Omron CX-Programmer project NewProject (CX-Programmer 9.74)

# PLC M1: CJ2M CPU32
I/O table (CPU CJ2M-CPU32): rack 0 slot 0 CJ1W-ID211; rack 0 slot 1 CJ1W-ID211; rack 0 slot 2 CJ1W-OD212; rack 0 slot 3 CJ1W-OC211; rack 0 slot 4 CJ1W-TC104; rack 0 slot 11 CJ2M-EIP21

## Data types
TYPE s_maquina_in : STRUCT  (* Inputs da maquina *)
  st_ciclo : BOOL;  (* Botão inicio de ciclo *)
  sp_ciclo : BOOL;  (* Botão fim de ciclo *)
  sel_carga : BOOL;  (* Botão selecção de carga *)
  st_carga : BOOL;  (* Botão inicio de carga *)
  fcf_carga : BOOL;  (* Fim de curso fechado carga *)
  sel_dcarga : BOOL;  (* Botão selecção de descarga *)
  st_dcarga : BOOL;  (* Botão inicio de descarga *)
  fcf_dcarga : BOOL;  (* Fim de curso fechado descarga *)
  psl : BOOL;  (* Pressostato *)
  nhrz : BOOL;  (* Maquina não horizontal *)
  pe1 : BOOL;  (* Paragem de emergência *)
  pe2 : BOOL;  (* Relé de segurança *)
  de : BOOL;  (* Disparo termico *)
  x0_13 : BOOL;  (* RESERVA *)
  x0_14 : BOOL;  (* RESERVA *)
  x0_15 : BOOL;  (* RESERVA *)
END_STRUCT END_TYPE
TYPE s_maquina_out : STRUCT  (* Outputs da maquina *)
  x0_0 : BOOL;  (* RESERVA *)
  x0_1 : BOOL;  (* RESERVA *)
  oma_carga : BOOL;  (* Abrir carga *)
  omf_carga : BOOL;  (* Fechar carga *)
  oma_dcarga : BOOL;  (* Abrir descarga *)
  omf_dcarga : BOOL;  (* Fechar descarga *)
  ok_carga : BOOL;  (* Carga confirmada (carregar rolhas) *)
  ok_dcarga : BOOL;  (* Descarga confirmada (descarregar rolhas) *)
  x0_8 : BOOL;  (* RESERVA *)
  x0_9 : BOOL;  (* RESERVA *)
  x0_10 : BOOL;  (* RESERVA *)
  x0_11 : BOOL;  (* RESERVA *)
  x0_12 : BOOL;  (* RESERVA *)
  x0_13 : BOOL;  (* RESERVA *)
  x0_14 : BOOL;  (* RESERVA *)
  x0_15 : BOOL;  (* RESERVA *)
END_STRUCT END_TYPE
TYPE s_maquina_lmp : STRUCT  (* Lampadas da maquina *)
  oms_inicio : BOOL;  (* Lampada inicio *)
  oms_carga : BOOL;  (* Lampada carga *)
  oms_dcarga : BOOL;  (* Lampada descarga *)
  x0_3 : BOOL;  (* RESERVA *)
  x0_4 : BOOL;  (* RESERVA *)
  x0_5 : BOOL;  (* RESERVA *)
  x0_6 : BOOL;  (* RESERVA *)
  x0_7 : BOOL;  (* RESERVA *)
  oms_red : BOOL;  (* Lampada FLASH vermelho *)
  oms_green : BOOL;  (* Lampada FLASH verde *)
  x0_10 : BOOL;  (* RESERVA *)
  x0_11 : BOOL;  (* RESERVA *)
  x0_12 : BOOL;  (* RESERVA *)
  x0_13 : BOOL;  (* RESERVA *)
  oms_ilum : BOOL;  (* Iluminação *)
  alm : BOOL;  (* Maquina em alarme (Alarmes que não páram a maquina) *)
END_STRUCT END_TYPE
TYPE s_maquina_defs : STRUCT  (* Defeitos da maquina *)
  def1 : BOOL;  (* Paragem de emergência *)
  def2 : BOOL;  (* Relé de segurança *)
  def3 : BOOL;  (* Disparo termico *)
  def4 : BOOL;  (* RESERVA *)
  def5 : BOOL;  (* Defeito de aspiração *)
  def6 : BOOL;  (* Defeito de tratamento *)
  def7 : BOOL;  (* Defeito de injecção *)
  def8 : BOOL;  (* Defeito de aquecimento *)
  def9 : BOOL;  (* Maquina não horizontal *)
  def10 : BOOL;  (* Pressão de ar baixa *)
  def11 : BOOL;  (* RESERVA *)
  def12 : BOOL;  (* RESERVA *)
  def13 : BOOL;  (* RESERVA *)
  def14 : BOOL;  (* RESERVA *)
  def15 : BOOL;  (* Falha de manobra na carga *)
  def16 : BOOL;  (* Falha de manobra na descarga *)
END_STRUCT END_TYPE
TYPE s_maquina_bits : STRUCT  (* Bits auxiliares da maquina *)
  rst : BOOL;  (* Reset aos defeitos *)
  dgm : BOOL;  (* Defeito geral *)
  mdp : BOOL;  (* Maquina disponivel *)
  x0_3 : BOOL;  (* RESERVA *)
  x0_4 : BOOL;  (* RESERVA *)
  x0_5 : BOOL;  (* RESERVA *)
  x0_6 : BOOL;  (* RESERVA *)
  x0_7 : BOOL;  (* RESERVA *)
  dp_tcarga : BOOL;  (* Transporte de carga disponivel (Maquina permite fazer transporte de carga) *)
  om_carga : BOOL;  (* Abrir carga *)
  om_dcarga : BOOL;  (* Abrir descarga *)
  LockDescarga : BOOL;  (* Bloquear descarga *)
  x0_12 : BOOL;  (* RESERVA *)
  x0_13 : BOOL;  (* RESERVA *)
  x0_14 : BOOL;  (* RESERVA *)
  x0_15 : BOOL;  (* RESERVA *)
  x1_0 : BOOL;  (* RESERVA *)
  x1_1 : BOOL;  (* RESERVA *)
  x1_2 : BOOL;  (* RESERVA *)
  x1_3 : BOOL;  (* RESERVA *)
  x1_4 : BOOL;  (* RESERVA *)
  x1_5 : BOOL;  (* RESERVA *)
  x1_6 : BOOL;  (* RESERVA *)
  inj_block : BOOL;  (* Injecção bloqueada *)
  act_ciclo : BOOL;  (* Ciclo - Activo *)
  om_ciclo : BOOL;  (* Ciclo - Ordem de marcha *)
  new_of : BOOL;  (* Nova ordem de fabrico *)
  val_ciclo : BOOL;  (* Ciclo validado pelo MES *)
  com_fail : BOOL;  (* Falha de comunicação com o MES *)
  st_mes : BOOL;  (* Arranque da ordem com MES *)
  x1_14 : BOOL;  (* RESERVA *)
  new_man : BOOL;  (* Nova ordem manual *)
END_STRUCT END_TYPE
TYPE s_maquina_hmi : STRUCT  (* Dados do HMI *)
  st_ciclo : BOOL;  (* Botão inicio de ciclo *)
  sp_ciclo : BOOL;  (* Botão fim de ciclo *)
  sel_carga : BOOL;  (* Botão selecção de carga *)
  st_carga : BOOL;  (* Botão inicio de carga *)
  sel_dcarga : BOOL;  (* Botão selecção de descarga *)
  st_dcarga : BOOL;  (* Botão inicio de descarga *)
  on_msg : BOOL;  (* Mostra janela de mensagens *)
  x0_7 : BOOL;  (* RESERVA *)
  x0_8 : BOOL;  (* RESERVA *)
  x0_9 : BOOL;  (* RESERVA *)
  x0_10 : BOOL;  (* RESERVA *)
  x0_11 : BOOL;  (* RESERVA *)
  x0_12 : BOOL;  (* RESERVA *)
  x0_13 : BOOL;  (* RESERVA *)
  x0_14 : BOOL;  (* RESERVA *)
  x0_15 : BOOL;  (* RESERVA *)
END_STRUCT END_TYPE
TYPE s_maquina : STRUCT  (* Dados da maquina *)
  modo : INT;  (* Modo de funcionamento (0-Manual, 1-Offline, 2-Online) *)
  etapa : INT;  (* Etapa actual (10-Carga, 20-Tratamento, 30-Descarga) *)
  in : s_maquina_in;  (* Entradas *)
  out : s_maquina_out;  (* Saidas *)
  hmi : s_maquina_hmi;  (* Dados do HMI *)
  bits : s_maquina_bits;  (* Bits auxiliares *)
  lmp : s_maquina_lmp;  (* Lampadas *)
  def : s_maquina_defs;  (* Defeitos *)
  cp_mes : s_maquina_mes;  (* Causas de paragem do MES *)
  log : s_maq_log;  (* Dados de datalogger *)
  pss_exe : s_pss_exe;  (* Passo actual a executar *)
  modo_hmi : INT;  (* Valor colocado pelo operador *)
  cparagem : INT;  (* Causa de paragem *)
  num_msg : INT;  (* Numero da mensagem *)
  rsv2 : INT Dimensions=[17];  (* RESERVA *)
  pt_sb : INT Dimensions=[5];  (* Zona SB da consola *)
  pt_sw : INT Dimensions=[5];  (* Zona SW da consola *)
END_STRUCT END_TYPE
TYPE s_f_aspira : STRUCT  (* Dados da função aspiração *)
  fca : BOOL;  (* Aspiração aberta *)
  fcf : BOOL;  (* Aspiração fechada *)
  oma : BOOL;  (* Abrir aspiração *)
  omf : BOOL;  (* Fechar aspiração *)
  rm : BOOL;  (* Resposta de marcha do ventilador de aspiração *)
  fm : BOOL;  (* Falha de manobra na aspiração *)
  fmv : BOOL;  (* Falha do ventilador de aspiração *)
  om_aquece : BOOL;  (* Aquecimento em curso (Pede aspiração) *)
  on : BOOL;  (* Aspiração em marcha e ok *)
  x0_9 : BOOL;  (* RESERVA *)
  x0_10 : BOOL;  (* RESERVA *)
  x0_11 : BOOL;  (* RESERVA *)
  x0_12 : BOOL;  (* RESERVA *)
  st_hmi : BOOL;  (* Arranque do hmi *)
  sp_hmi : BOOL;  (* Paragem do hmi *)
  cfm : BOOL;  (* Condição de funcionamento manual *)
  es : INT;  (* Estado *)
  rsv1 : INT Dimensions=[16];  (* RESERVA *)
  tt : REAL;  (* Totalizador *)
END_STRUCT END_TYPE
TYPE s_tc104_cio : STRUCT  (* Dados CIO da carta TC104 *)
  sp1 : INT;  (* Loop 1 Set Point (SP) *)
  sp2 : INT;  (* Loop 2 Set Point (SP) *)
  l2_st_at : BOOL;  (* Loop 2 Start AT *)
  l2_sp_at : BOOL;  (* Loop 2 Stop AT *)
  l1_st_at : BOOL;  (* Loop 1 Start AT *)
  l1_sp_at : BOOL;  (* Loop 1 Stop AT *)
  l2_sp : BOOL;  (* Loop 2 Stop *)
  x2_5 : BOOL;  (* RESERVA *)
  l1_sp : BOOL;  (* Loop 1 Stop *)
  x2_7 : BOOL;  (* RESERVA *)
  x2_8 : BOOL;  (* RESERVA *)
  x2_9 : BOOL;  (* RESERVA *)
  x2_10 : BOOL;  (* RESERVA *)
  x2_11 : BOOL;  (* RESERVA *)
  l2_ch_pid_c : BOOL;  (* Loop 2 Change PID Constants *)
  l1_ch_pid_c : BOOL;  (* Loop 1 Change PID Constants *)
  l2_save : BOOL;  (* Loop 2 Save *)
  l1_save : BOOL;  (* Loop 1 Save *)
  pv1 : INT;  (* Loop 1 PV *)
  pv2 : INT;  (* Loop 2 PV *)
  sp1_r : INT;  (* Loop 1 Set Point (SP) - Read *)
  sp2_r : INT;  (* Loop 2 Set Point (SP) - Read *)
  l1_l2_dp_err : WORD;  (* Loop 1/2 Decimal point & error number *)
  l1_s_al2 : BOOL;  (* Loop 1 - Status AL2 *)
  l1_s_al1 : BOOL;  (* Loop 1 - Status AL1 *)
  l1_s_hb : BOOL;  (* Loop 1 - Status HB *)
  l1_s_at : BOOL;  (* Loop 1 - Status AT *)
  l1_s_ctrlout : BOOL;  (* Loop 1 - Status Control Output *)
  x8_5 : BOOL;  (* RESERVA *)
  x8_6 : BOOL;  (* RESERVA *)
  x8_7 : BOOL;  (* RESERVA *)
  l1_s_sp : BOOL;  (* Loop 1 - Status Stop *)
  l1_s_err : BOOL;  (* Loop 1 - Status Setting Error *)
  l1_s_pid_calc : BOOL;  (* Loop 1 - Status PID Constants Calculated *)
  l1_s_sby : BOOL;  (* Loop 1 - Status Standby *)
  l1_s_ferr : BOOL;  (* Loop 1 - Status Fatal Error *)
  l1_s_ct_ovf : BOOL;  (* Loop 1 - Status Overflow *)
  l1_s_serr : BOOL;  (* Loop 1 - Status Sensor Error *)
  l1_s_savec : BOOL;  (* Loop 1 - Status Save Completed *)
  l2_s_al2 : BOOL;  (* Loop 2 - Status AL2 *)
  l2_s_al1 : BOOL;  (* Loop 2 - Status AL1 *)
  l2_s_hb : BOOL;  (* Loop 2 - Status HB *)
  l2_s_at : BOOL;  (* Loop 2 - Status AT *)
  l2_s_ctrlout : BOOL;  (* Loop 2 - Status Control Output *)
  x9_5 : BOOL;  (* RESERVA *)
  x9_6 : BOOL;  (* RESERVA *)
  x9_7 : BOOL;  (* RESERVA *)
  l2_s_sp : BOOL;  (* Loop 2 - Status Stop *)
  l2_s_err : BOOL;  (* Loop 2 - Status Setting Error *)
  l2_s_pid_calc : BOOL;  (* Loop 2 - Status PID Constants Calculated *)
  l2_s_sby : BOOL;  (* Loop 2 - Status Standby *)
  l2_s_ferr : BOOL;  (* Loop 2 - Status Fatal Error *)
  l2_s_ct_ovf : BOOL;  (* Loop 2 - Status Overflow *)
  l2_s_serr : BOOL;  (* Loop 2 - Status Sensor Error *)
  l2_s_savec : BOOL;  (* Loop 2 - Status Save Completed *)
  hb_sp1 : INT;  (* Loop 1 - Heater Burnout Set Value *)
  hb_sp2 : INT;  (* Loop 2 - Heater Burnout Set Value *)
  rsv1 : INT;  (* RESERVA *)
  hc1 : INT;  (* Loop 1 - Heater Current *)
  hc2 : INT;  (* Loop 2 - Heater Current *)
  hb_sp1_r : INT;  (* Loop 1 - Heater Burnout Set Value - Read *)
  hb_sp2_r : INT;  (* Loop 2 - Heater Burnout Set Value - Read *)
  rsv2 : INT Dimensions=[3];  (* RESERVA *)
END_STRUCT END_TYPE
TYPE s_tc104_dm : STRUCT  (* Dados DM da carta TC104 *)
  dados : INT Dimensions=[100];  (* Dados da carta *)
END_STRUCT END_TYPE
TYPE s_f_aquece : STRUCT  (* Dados da função aquecimento *)
  rm_r : BOOL;  (* Contactor das resistências *)
  rm_v : BOOL;  (* Resposta de marcha do ventilador *)
  ok_fx : BOOL;  (* Detector de fluxo OK *)
  x0_3 : BOOL;  (* RESERVA *)
  ft : BOOL;  (* Falha de temperatura *)
  ini : BOOL;  (* Inicio do aquecimento *)
  ini_tt : BOOL;  (* Inicio da contagem do tempo *)
  ok_sp : BOOL;  (* Dentro da vizinhaça de setpoint a controlar *)
  om : BOOL;  (* Ordem de marcha para aquecimento *)
  fm_r : BOOL;  (* Falha de marcha das resistências *)
  fm_v : BOOL;  (* Falha de marcha do ventilador *)
  fm_fx : BOOL;  (* Falha no detector de fluxo *)
  fm_a : BOOL;  (* Falha na aspiração *)
  st_hmi : BOOL;  (* Arranque do hmi *)
  sp_hmi : BOOL;  (* Paragem do hmi *)
  cfm : BOOL;  (* Condição de funcionamento manual *)
  es_r : INT;  (* Estado *)
  sp : REAL;  (* Setpoint de temperatura *)
  pv : REAL;  (* Temperatura actual *)
  sp_delta : REAL;  (* Valor de vizinhança apartir do qual começa a contar tempo de aquecimento *)
  sp_ft : INT;  (* Tempo para dar falha de temperatura *)
  es_v : INT;  (* Estado *)
  rsv2 : INT Dimensions=[8];  (* RESERVA *)
  tt : REAL;  (* Totalizador *)
END_STRUCT END_TYPE
TYPE s_f_trata : STRUCT  (* Dados da função tratamento *)
  rm : BOOL;  (* Marcha do tambor *)
  om1 : BOOL;  (* Ordem de marcha 1 *)
  om2 : BOOL;  (* Ordem de marcha 2 *)
  omx : BOOL;  (* Ordem de marcha auxiliar *)
  fm : BOOL;  (* Falha de marcha do tambor *)
  x0_5 : BOOL;  (* RESERVA *)
  x0_6 : BOOL;  (* RESERVA *)
  x0_7 : BOOL;  (* RESERVA *)
  x0_8 : BOOL;  (* RESERVA *)
  x0_9 : BOOL;  (* RESERVA *)
  x0_10 : BOOL;  (* RESERVA *)
  x0_11 : BOOL;  (* RESERVA *)
  x0_12 : BOOL;  (* RESERVA *)
  x0_13 : BOOL;  (* RESERVA *)
  x0_14 : BOOL;  (* RESERVA *)
  cfm : BOOL;  (* Condição de funcionamento manual *)
  es : INT;  (* Estado *)
  rsv2 : INT Dimensions=[16];  (* RESERVA *)
  tt : REAL;  (* Totalizador *)
END_STRUCT END_TYPE
TYPE s_f_injecta : STRUCT  (* Dados da função injecção *)
  x0_0 : BOOL;  (* RESERVA *)
  x0_1 : BOOL;  (* RESERVA *)
  om1 : BOOL;  (* Ordem de marcha *)
  om2 : BOOL;  (* Ordem de marcha spray *)
  finj : BOOL;  (* Falha de injecção *)
  fg : BOOL;  (* Fuga de produto *)
  x0_6 : BOOL;  (* RESERVA *)
  s_insp : BOOL;  (* Inspecção activada *)
  inj : BOOL;  (* Pede permissão para injectar *)
  inj_ok : BOOL;  (* Recebe autorização para injectar *)
  x0_10 : BOOL;  (* RESERVA *)
  x0_11 : BOOL;  (* RESERVA *)
  x0_12 : BOOL;  (* RESERVA *)
  x0_13 : BOOL;  (* RESERVA *)
  cal : BOOL;  (* Calibração *)
  cfm : BOOL;  (* Condição de funcionamento manual *)
  es : INT;  (* Estado *)
  prod : INT;  (* Produto *)
  rsv1 : INT Dimensions=[15];  (* RESERVA *)
  tt : REAL;  (* Totalizador *)
END_STRUCT END_TYPE
TYPE s_caudal : STRUCT  (* Dados do caudalimetro *)
  tti : BOOL;  (* Impulso de totalização *)
  rst : BOOL;  (* Reset *)
  prod_used : BOOL;  (* Produto em uso *)
  fgp : BOOL;  (* Fuga de produto *)
  ftt : BOOL;  (* Falha de caudal *)
  rem : BOOL;  (* Totalizador local/remoto *)
  rem_ok : BOOL;  (* OK para ir buscar o valor do totalizador remoto *)
  inj_ini : BOOL;  (* Inicio da injecção *)
  x0_8 : BOOL;  (* RESERVA *)
  x0_9 : BOOL;  (* RESERVA *)
  x0_10 : BOOL;  (* RESERVA *)
  x0_11 : BOOL;  (* RESERVA *)
  x0_12 : BOOL;  (* RESERVA *)
  x0_13 : BOOL;  (* RESERVA *)
  x0_14 : BOOL;  (* RESERVA *)
  x0_15 : BOOL;  (* RESERVA *)
  prod : INT;  (* Produto *)
  rsv1 : INT Dimensions=[6];  (* RESERVA *)
  tti_x : REAL;  (* Valor do impulso *)
  tt_rem : REAL;  (* Totalizador remoto *)
  tt_rem_old : REAL;  (* Totalizador remoto antigo *)
  tt_inj : REAL;  (* Totalizador de injecção *)
  tt_p : REAL;  (* Totalizador parcial *)
  tt_g : REAL;  (* Totalizador global *)
END_STRUCT END_TYPE
TYPE s_carro : STRUCT  (* Dados do carro de injecção *)
  fcr : BOOL;  (* Fim de curso recuado *)
  fca : BOOL;  (* Fim de curso avanço *)
  oma : BOOL;  (* Ordem de marcha avanço *)
  omr : BOOL;  (* Ordem de marcha recuar *)
  omv : BOOL;  (* Ordem de marcha velocidade lenta *)
  fm : BOOL;  (* Falha de manobra *)
  av : BOOL;  (* Avaria *)
  i_pos : BOOL;  (* Impulsos de posição *)
  inj : BOOL;  (* Recebe pedido para injectar *)
  inj_ok : BOOL;  (* Informa que pode injectar *)
  cal : BOOL;  (* Calibrar *)
  src : BOOL;  (* Sentido recuar *)
  dgm : BOOL;  (* Defeito geral de maquina *)
  rm : BOOL;  (* Resposta de marcha *)
  cfma : BOOL;  (* Condição de funcionamento manual avançar *)
  cfmr : BOOL;  (* Condição de funcionamento manual recuar *)
  fav : BOOL;  (* Falha por avaria *)
  s_dp : BOOL;  (* Carrinho habilitado *)
  inj_cal : BOOL;  (* Calibração da injecção *)
  s_aut : BOOL;  (* Automatico *)
  x1_4 : BOOL;  (* RESERVA *)
  x1_5 : BOOL;  (* RESERVA *)
  x1_6 : BOOL;  (* RESERVA *)
  x1_7 : BOOL;  (* RESERVA *)
  x1_8 : BOOL;  (* RESERVA *)
  x1_9 : BOOL;  (* RESERVA *)
  x1_10 : BOOL;  (* RESERVA *)
  x1_11 : BOOL;  (* RESERVA *)
  x1_12 : BOOL;  (* RESERVA *)
  x1_13 : BOOL;  (* RESERVA *)
  x1_14 : BOOL;  (* RESERVA *)
  x1_15 : BOOL;  (* RESERVA *)
  rsv1 : INT Dimensions=[10];  (* RESERVA *)
  sp_min : REAL;  (* Setpoint posição minima de injecção *)
  sp_max : REAL;  (* Setpoint posição maxima de injecção *)
  pos_act : REAL;  (* Posição actual *)
  tt_i_act : INT;  (* Numero de impulsos actuais *)
  tt_i_max : INT;  (* Numero de impulsos maximos *)
END_STRUCT END_TYPE
TYPE s_of_cliente : STRUCT  (* Dados do cliente de uma OF *)
  nome : WORD Dimensions=[25];  (* Nome do cliente *)
  data : WORD Dimensions=[10];  (* Data de entrega *)
  produto : WORD Dimensions=[20];  (* Nome do produto *)
  prg_on : WORD Dimensions=[5];  (* Numero do programa online *)
  n_enc : WORD Dimensions=[10];  (* Numero de encomenda *)
  n_of : WORD Dimensions=[10];  (* Numero da OF *)
  n_lt : WORD Dimensions=[10];  (* Numero do lote *)
END_STRUCT END_TYPE
TYPE s_of_totais : STRUCT  (* Totais produzidos e a produzir de uma OF *)
  tt_global : UDINT;  (* Total a produzir na OF *)
  tt_falta : UDINT;  (* Total que falta produzir na OF *)
  tt_produzir : UDINT;  (* Total a produzir na maquina no batch *)
END_STRUCT END_TYPE
TYPE s_of_calibre : STRUCT  (* Calibre das rolhas a usar na OF *)
  dmt1 : REAL;  (* Diametro da rolha *)
  dmt2 : REAL;  (* Diametro da rolha *)
  h : REAL;  (* Comprimento da rolha *)
  a : REAL;  (* Area da rolha *)
  qtp : REAL;  (* Quantidade de produto *)
  cl_txt : WORD Dimensions=[10];  (* Calibre - Texto *)
END_STRUCT END_TYPE
TYPE s_of_pss : STRUCT  (* Passo individual do programa a executar *)
  f : INT;  (* Função *)
  p1 : INT;  (* Parametro 1 *)
  p2 : REAL;  (* Parametro 2 *)
  tt : REAL;  (* Totalizador *)
  uni : INT;  (* Unidade do totalizador *)
  rsv : INT Dimensions=[3];  (* RESERVA *)
END_STRUCT END_TYPE
TYPE s_of_prg : STRUCT  (* Programa a ser executado *)
  pss : s_of_pss Dimensions=[12];  (* Passos do programa a executar *)
END_STRUCT END_TYPE
TYPE s_of : STRUCT  (* Ordem de fabrico *)
  cliente : s_of_cliente;  (* Cliente da OF *)
  totais : s_of_totais;  (* Totais da OF *)
  calibre : s_of_calibre;  (* Calibre das rolhas da OF *)
  dados : BOOL;  (* OF com valores *)
  online : BOOL;  (* Ordem com dados para funcionar online *)
  nprg_off : INT;  (* Numero do programa offline *)
  rsv1 : INT Dimensions=[8];  (* RESERVA *)
  prg : s_of_prg;  (* Programa *)
END_STRUCT END_TYPE
TYPE s_pss_exe : STRUCT  (* Passo a executar *)
  pss : s_of_pss;  (* Passo actual a executar *)
  num_pss : INT;  (* Numero do passo actual *)
  ini : BOOL;  (* Inicio - Inicio do passo (Função faz inicializações necessárias) *)
  exe : BOOL;  (* Executar - Condição para funcionar (Função actua se valor igual a 1) *)
  fim : BOOL;  (* Fim - Terminado o passo (Função indica que terminou de executar) *)
  exc : BOOL;  (* Exclusivo - Condição para funções exclusivas (Função exclusiva coloca a 0 ao executar, impedindo que outras o façam) *)
  log : BOOL;  (* Fazer log *)
  rsv1 : INT Dimensions=[8];  (* RESERVA *)
END_STRUCT END_TYPE
TYPE s_mes_com : STRUCT  (* Comunicação com o MES *)
  n_enc : WORD Dimensions=[10];  (* Numero de encomenda *)
  n_of : WORD Dimensions=[10];  (* Numero da OF *)
  n_lt : WORD Dimensions=[10];  (* Numero do lote *)
  user : WORD Dimensions=[10];  (* Codigo do operador *)
  rsv1 : INT;  (* RESERVA *)
  mes_plc : INT;  (* Variável de verificação de comunicação do MES para o PLC *)
  mes_plcx : INT;  (* Variável de verificação de comunicação do MES para o PLC (Auxiliar) *)
  plc_mes : INT;  (* Variável de verificação de comunicação do PLC para o MES *)
  mes_com_fail : BOOL;  (* Falha de comunicação com o MES *)
  f_in_exe : INT;  (* Função a executar *)
  f_out_exe : INT;  (* Função executada *)
  new_of : INT;  (* Contador de nova OF *)
  ctrl_com_plc : INT;  (* Controlo da comunicação - Escrita do PLC *)
  ctrl_com_mes : INT;  (* Controlo da comunicação - Escrita do MES *)
END_STRUCT END_TYPE
TYPE s_maq_log : STRUCT  (* Dados de datalogger da maquina *)
  n_of : WORD Dimensions=[10];  (* Numero da OF *)
  user : WORD Dimensions=[10];  (* Codigo do operador *)
  pss_exe : s_pss_exe;  (* Dados do passo actual *)
END_STRUCT END_TYPE
TYPE s_maquina_mes : STRUCT  (* Causas de paragem para o MES *)
  cp8 : BOOL;  (* Problemas de caudal *)
  cp9 : BOOL;  (* Filtro entupido *)
  cp10 : BOOL;  (* Bomba desligada *)
  cp11 : BOOL;  (* Obstrução da linha *)
  cp6 : BOOL;  (* Alarme de aquecimento *)
  cp13 : BOOL;  (* Falha de sonda *)
  cp19 : BOOL;  (* Descarga sem tratamento *)
  cp5 : BOOL;  (* Falta de tensão *)
  cp15 : BOOL;  (* Fuga de produto *)
  cp18 : BOOL;  (* Baixa temperatura *)
  cp7 : BOOL;  (* Falha geral *)
  X0_11 : BOOL;  (* RESERVA *)
  x0_12 : BOOL;  (* RESERVA *)
  x0_13 : BOOL;  (* RESERVA *)
  x0_14 : BOOL;  (* RESERVA *)
  x0_15 : BOOL;  (* RESERVA *)
END_STRUCT END_TYPE
TYPE s_equip_ios : STRUCT  (* Equipamento - Entradas *)
  om : BOOL;  (* Ordem de marcha *)
  oma : BOOL;  (* Ordem de abrir *)
  omf : BOOL;  (* Ordem de fechar *)
  rm : BOOL;  (* Resposta de marcha *)
  fca : BOOL;  (* Fim de curso aberta *)
  fcf : BOOL;  (* Fim de curso fechada *)
  de : BOOL;  (* Defeito electrico *)
  pf_bmb : BOOL;  (* Pulsos de funcionamento da bomba *)
END_STRUCT END_TYPE
TYPE s_equip_bits : STRUCT  (* Equipamento - Bits auxiliares *)
  s_aut : BOOL;  (* Automatico *)
  mdp : BOOL;  (* Disponibilidade *)
  ndp : BOOL;  (* Não disponivel *)
  dgm : BOOL;  (* Defeito geral de maquina *)
  rst : BOOL;  (* Reset *)
  cfa : BOOL;  (* Condição de funcionamento automatico *)
  cfm : BOOL;  (* Condição de funcionamento manual *)
  cfaa : BOOL;  (* Condição de funcionamento automatico abrir *)
  cfaf : BOOL;  (* Condição de funcionamento automatico fechar *)
  cfma : BOOL;  (* Condição de funcionamento manual abrir *)
  cfmf : BOOL;  (* Condição de funcionamento manual fechar *)
  st_hmi : BOOL;  (* Arranque HMI *)
  sp_hmi : BOOL;  (* Paragem HMI *)
  p_hmi : BOOL;  (* Pausa HMI *)
END_STRUCT END_TYPE
TYPE s_equip_defs : STRUCT  (* Equipamentos - Defeitos *)
  fm : BOOL;  (* Falha de marcha *)
  fma : BOOL;  (* Falha de manobra abrir *)
  fmf : BOOL;  (* Falha de manobra fechar *)
  de : BOOL;  (* Defeito electrico *)
  dv : BOOL;  (* Deposito vazio *)
END_STRUCT END_TYPE
TYPE s_equip : STRUCT  (* Equipamento *)
  ios : s_equip_ios;  (* Entradas *)
  bits : s_equip_bits;  (* Bits *)
  defs : s_equip_defs;  (* Defeitos *)
  es : INT;  (* Estado *)
  tm_b : INT;  (* Tempo entre bombagens *)
  rsv1 : INT Dimensions=[5];  (* Reserva *)
END_STRUCT END_TYPE
TYPE s_Steps : STRUCT
  f : INT;  (* Função *)
  p1 : INT;  (* Parametro 1 *)
  p2 : REAL;  (* Parametro 2 *)
END_STRUCT END_TYPE
TYPE s_Estado : STRUCT
  Ciclo : BOOL;  (* Em ciclo produtivo *)
  FimCiclo : BOOL;  (* Finalização ciclo *)
  Estado : BOOL;  (* Estado equipamento *)
  FimTratamento : BOOL;  (* Tratamento Finalizado *)
  OF_Carregada : BOOL;  (* Ordem carregada para máquina *)
  Avaria : BOOL;  (* Máquina em Avaria *)
  Com_OF : BOOL;  (* Máquina com OF carregada *)
  FalhaInjeProd : BOOL;  (* Falta de injeção de produto *)
  FalhaAquecim : BOOL;  (* Falha de aquecimento *)
  AvariaTermicos : BOOL;  (* Avaria de térmicos *)
  TratAbortado : BOOL;  (* Tratamento abortado pelo operador *)
  FalhaEnergia : BOOL;  (* Falha energia *)
  NivelProdBaixo : BOOL;  (* Nível produto químico no depósito baixo *)
  Manual : BOOL;  (* modo manual *)
  Emergencia : BOOL;  (* Paragem Emergência *)
END_STRUCT END_TYPE

## Global symbols (name address type ; comment)
Exe_Time ExeTimeCalc
Steps_Copy fb_CopySteps
bit_Injecao W500.05 BOOL
fb_inj_caudal_01 fb_inj_caudal
fb_inj_caudal_02 fb_inj_caudal
fb_inj_caudal_03 fb_inj_caudal
fb_inj_caudal_04 fb_inj_caudal
fb_inj_caudal_05 fb_inj_caudal
fb_m fb_maquina
fb_m_f_aquece fb_f_aquece
fb_m_f_aspira fb_f_aspira
fb_m_f_injecta1 fb_f_injecta
fb_m_f_injecta2 fb_f_injecta
fb_m_f_injecta3 fb_f_injecta
fb_m_f_injecta4 fb_f_injecta
fb_m_f_injecta5 fb_f_injecta
fb_m_f_injecta_man fb_f_injecta_man
fb_m_f_trata fb_f_trata
fb_m_mes_com_trp fb_mes_com_trp
fb_maquina_pss_2_str10 fb_maquina_pss_2_str10_PT
fb_maquina_pss_2_str10_off fb_maquina_pss_2_str10_PT
fb_mes_cparagem fb_mes_cparagem
oms_ilum 3.07 BOOL  ; Iluminação

## Program Maquina (cyclic task 0)
Local symbols
BatchReal E0_5100 STRUCT s_Steps
Cnt_Inv W508 REAL
Estado E0_5107 STRUCT s_Estado
ExeCDT D4631 INT
ExeTotalTime D4630 INT
M_Online W100.05 BOOL
Receita_Maq E0_5000 STRUCT[12] s_Steps
Receita_Maq_Ok E0_5048.00 BOOL
Temperatura E0_5105 INT
TranspDest E0_5106 UINT
bit_Aquecimento W500.03 BOOL
bit_Aspiracao W500.02 BOOL
bit_Carga W500.00 BOOL
bit_Descarga W500.01 BOOL
bit_FCiclo W100.04 BOOL
bit_FimDCarga W500.06 BOOL
bit_Tratamento W500.04 BOOL
de_carro 1.10 BOOL  ; Avaria conversor carrinho
de_m 0.12 BOOL  ; Disparo magnetotermicos
fc_nhrz 1.08 BOOL  ; Maquina não horizontal
fca_aspira 1.09 BOOL  ; Aspiração aberta
fca_carga 1.06 BOOL  ; Porta carga aberta
fca_carro 1.14 BOOL  ; $?St$Bk?_#[39] / Carrinho na posição "frente"$?St$Bk?_#[39]
fcf_dcarga 1.07 BOOL  ; Porta descarga fechada
fcr_carro 1.13 BOOL  ; $?St$Bk?_#[40] / Carrinho na posição "zero"$?St$Bk?_#[40]
ft01 D700 STRUCT s_caudal  ; Caudalímetro
ft02 D720 STRUCT s_caudal  ; Caudalímetro
ft03 D740 STRUCT s_caudal  ; Caudalímetro
ft04 D760 STRUCT s_caudal  ; Caudalímetro
ft05 D780 STRUCT s_caudal  ; Caudalímetro
m D0 STRUCT s_maquina  ; Maquina - Maquina
m1_dlog_fifo_1 E130 STRING[130]
m1_dlog_fifo_10 E1300 STRING[130]
m1_dlog_fifo_11 E1430 STRING[130]
m1_dlog_fifo_12 E1560 STRING[130]
m1_dlog_fifo_13 E1690 STRING[130]
m1_dlog_fifo_2 E260 STRING[130]
m1_dlog_fifo_3 E390 STRING[130]
m1_dlog_fifo_4 E520 STRING[130]
m1_dlog_fifo_5 E650 STRING[130]
m1_dlog_fifo_6 E780 STRING[130]
m1_dlog_fifo_7 E910 STRING[130]
m1_dlog_fifo_8 E1040 STRING[130]
m1_dlog_fifo_9 E1170 STRING[130]
m1_dlog_fifo_in E0 STRING[130]
m1_dlog_fifo_out E1820 STRING[130]
m_dlog_event_file_name W125 STRING[8]  ; Nome do ficheiro de datalogger
m_dlog_event_read W100.01 BOOL  ; Bit para apagar datalogger
m_dlog_event_value W102 REAL  ; Valor para o datalogger
m_dlog_hum_file_name W135 STRING[8]  ; Nome do ficheiro de datalogger
m_dlog_hum_read W100.03 BOOL  ; Bit para apagar datalogger
m_dlog_humid_value W106 REAL  ; Valor para o datalogger
m_dlog_maq_file_name W120 STRING[8]  ; Nome do ficheiro de datalogger
m_dlog_maq_name W110 STRING[10]  ; Nome da maquina
m_dlog_maq_read W100.00 BOOL  ; Bit para apagar datalogger
m_dlog_temp_file_name W130 STRING[8]  ; Nome do ficheiro de datalogger
m_dlog_temp_read W100.02 BOOL  ; Bit para apagar datalogger
m_dlog_temp_value W104 REAL  ; Valor para o datalogger
m_f10_as1 D500 STRUCT s_f_aspira  ; Maquina - Aspiração
m_f20_aq1 D520 STRUCT s_f_aquece  ; Maquina - Aquecimento
m_f30_tr1 D540 STRUCT s_f_trata  ; Maquina - Tratamento
m_f40_inj1 D560 STRUCT s_f_injecta  ; Maquina - Injecção 1
m_f40_inj2 D580 STRUCT s_f_injecta  ; Maquina - Injecção 2
m_f40_inj3 D600 STRUCT s_f_injecta  ; Maquina - Injecção 3
m_f40_inj4 D620 STRUCT s_f_injecta  ; Maquina - Injecção 4
m_f40_inj5 D640 STRUCT s_f_injecta  ; Maquina - Injecção 5
m_log_n_of D10 STRING[20]  ; Maquina - String do numero da OF para log
m_log_user D20 STRING[20]  ; Maquina - String do user para log
m_maq D0 STRUCT s_maquina
m_mes_com_exe D900 STRUCT s_mes_com  ; Comunicação com o MES (Tratamento)
m_mes_com_trp D950 STRUCT s_mes_com  ; Comunicação com o MES (Transporte)
m_of1_exe D1024 STRUCT s_of  ; Maquina - Dados da OF a ser executada
m_of2_maq D1274 STRUCT s_of  ; Maquina - Dados da OF carregados na maquina
m_of3_trp D1524 STRUCT s_of  ; Maquina - Dados da OF recebidos do transporte
m_str_act D170 STRING[30]  ; String do passo actual
m_str_off_prg0 D4300 STRING[10]  ; String do programa offline 0
m_str_off_prg1 D4310 STRING[10]  ; String do programa offline 1
m_str_off_prg10 D4400 STRING[10]  ; String do programa offline 10
m_str_off_prg11 D4410 STRING[10]  ; String do programa offline 11
m_str_off_prg12 D4420 STRING[10]  ; String do programa offline 12
m_str_off_prg13 D4430 STRING[10]  ; String do programa offline 13
m_str_off_prg14 D4440 STRING[10]  ; String do programa offline 14
m_str_off_prg2 D4320 STRING[10]  ; String do programa offline 2
m_str_off_prg3 D4330 STRING[10]  ; String do programa offline 3
m_str_off_prg4 D4340 STRING[10]  ; String do programa offline 4
m_str_off_prg5 D4350 STRING[10]  ; String do programa offline 5
m_str_off_prg6 D4360 STRING[10]  ; String do programa offline 6
m_str_off_prg7 D4370 STRING[10]  ; String do programa offline 7
m_str_off_prg8 D4380 STRING[10]  ; String do programa offline 8
m_str_off_prg9 D4390 STRING[10]  ; String do programa offline 9
m_str_off_pss0 D4000 STRING[30]  ; String do programa offline passo 0
m_str_off_pss1 D4030 STRING[30]  ; String do programa offline passo 1
m_str_off_pss10 D5060 STRING[30]  ; String do programa offline passo 10
m_str_off_pss11 D5090 STRING[30]  ; String do programa offline passo 11
m_str_off_pss2 D4060 STRING[30]  ; String do programa offline passo 2
m_str_off_pss3 D4090 STRING[30]  ; String do programa offline passo 3
m_str_off_pss4 D4120 STRING[30]  ; String do programa offline passo 4
m_str_off_pss5 D4150 STRING[30]  ; String do programa offline passo 5
m_str_off_pss6 D4180 STRING[30]  ; String do programa offline passo 6
m_str_off_pss7 D4210 STRING[30]  ; String do programa offline passo 7
m_str_off_pss8 D4240 STRING[30]  ; String do programa offline passo 8
m_str_off_pss9 D4270 STRING[30]  ; String do programa offline passo 9
m_str_pss0 D200 STRING[30]  ; String do passo 0
m_str_pss1 D230 STRING[30]  ; String do passo 1
m_str_pss10 D5000 STRING[30]  ; String do passo 10
m_str_pss11 D5030 STRING[30]  ; String do passo 11
m_str_pss2 D260 STRING[30]  ; String do passo 2
m_str_pss3 D290 STRING[30]  ; String do passo 3
m_str_pss4 D320 STRING[30]  ; String do passo 4
m_str_pss5 D350 STRING[30]  ; String do passo 5
m_str_pss6 D380 STRING[30]  ; String do passo 6
m_str_pss7 D410 STRING[30]  ; String do passo 7
m_str_pss8 D440 STRING[30]  ; String do passo 8
m_str_pss9 D470 STRING[30]  ; String do passo 9
m_tc104_cio 2000 STRUCT s_tc104_cio
m_tc104_dm D20000 STRUCT s_tc104_dm
maq_rz D690 STRUCT s_equip  ; Razeira da maquina
of_off_prg_num W200 INT  ; Programa a ser alterado offline
ok_fx_aquece 1.12 BOOL  ; Detector de fluxo OK
om2_fx_aquece 2.04 BOOL  ; Detector de fluxo
om2_injecta 2.12 BOOL  ; pistola 2
om2_tambor 2.01 BOOL  ; Rotação 2 tambor
om33_injecta 3.10 BOOL  ; Spray pistola 3
om34_injecta 3.11 BOOL  ; Spray pistola 4
om35_injecta 3.12 BOOL  ; Spray pistola 5
om3_injecta 2.13 BOOL  ; $?St$Bk?_#[41] / Pistola 3 / $?St$Bk?_#[41]
om4_injecta 2.14 BOOL  ; Pistola 4
om5_injecta 2.15 BOOL  ; Pistola 5
om_braco 3.09 BOOL  ; Braço basculante das pistolas
om_carro 3.13 BOOL  ; Carrinho RUN
om_injecta 2.11 BOOL  ; $?St$Bk?_#[42] / Pistola 1 / $?St$Bk?_#[42]
om_r_aquece 2.03 BOOL  ; Contactor 1 resistencias
om_tambor 2.00 BOOL  ; Rotação 1 tambor
om_v_aquece 2.02 BOOL  ; Ventilador de resistencias/detetor Fluxo
oma_aspira 2.05 BOOL  ; Valvula exaustão
oma_carga 2.06 BOOL  ; Porta carga/abre
oma_dcarga 2.08 BOOL  ; Porta descarga/abre
omf_carga 2.07 BOOL  ; Porta carga/fecha
omf_dcarga 2.09 BOOL  ; Porta descarga/fecha
omr_carro 3.15 BOOL  ; Carrinho reverse
oms_carga 3.01 BOOL  ; Lampada porta carga
oms_dcarga 3.02 BOOL  ; Lampada porta descarga
oms_green 3.05 BOOL  ; FLASH verde
oms_inicio 3.00 BOOL  ; Lampada inicio
oms_red 3.06 BOOL  ; FLASH vermelho
oms_tp1 3.03 BOOL  ; Lampada transporte 1
oms_tp2 3.04 BOOL  ; Lampada transporte 2
omv2_carro 3.14 BOOL  ; Carrinho velocidade 2
pe1_m 0.00 BOOL  ; Botão emergencia
pe2_m 0.15 BOOL  ; Sinal rele segurança activo
prg_exe D4500 STRUCT s_of_prg  ; Programa a executar
prg_off D2000 STRUCT[15] s_of_prg  ; Programas offline
prg_off_config D3700 STRUCT s_of_prg  ; Programa em configuração
prg_on D3850 STRUCT s_of_prg  ; Programa online
prod_used D10009.00 BOOL[10]  ; Produto em uso
psl_m 1.05 BOOL  ; Pressostato maquina
rm_carro 0.14 BOOL  ; Marcha carrinho
rm_r_aquece 0.11 BOOL  ; Confirmação contactor resistencias
rm_tambor 0.09 BOOL  ; Confirmação rotação
rm_v_aquece 0.10 BOOL  ; Confirmação contactor ventilador resistencias
sel_carga 0.03 BOOL  ; Selector carga( Abre porta carga)
sel_dcarga 0.05 BOOL  ; Selector descarga
sp_ciclo 0.02 BOOL  ; Botão stop ciclo
st_carga 0.04 BOOL  ; Botão confirma (Abre razeira moega)
st_ciclo 0.01 BOOL  ; Botão inicio ciclo
st_dcarga 0.06 BOOL  ; Botão confirma (Abre porta descarga)
st_sp_trp1 0.07 BOOL  ; Botão liga/desliga tapete descarga 1
st_sp_trp2 0.08 BOOL  ; Botão liga/desliga tapete descarga 2
str_data_hora H100 STRING[30]  ; String data/hora para datalogger
str_dummy D140 STRING[30]  ; String do auxiliar
tmp_Real W510 REAL
tt_carro 1.15 BOOL  ; Impulsos do carrinho
tti1 1.00 BOOL  ; Caudalimetro 1
tti2 1.01 BOOL  ; Caudalimetro 2
tti3 1.02 BOOL  ; Caudalimetro 3
tti4 1.03 BOOL  ; Caudalimetro 4
tti5 1.04 BOOL  ; Caudalimetro 5

### Section M

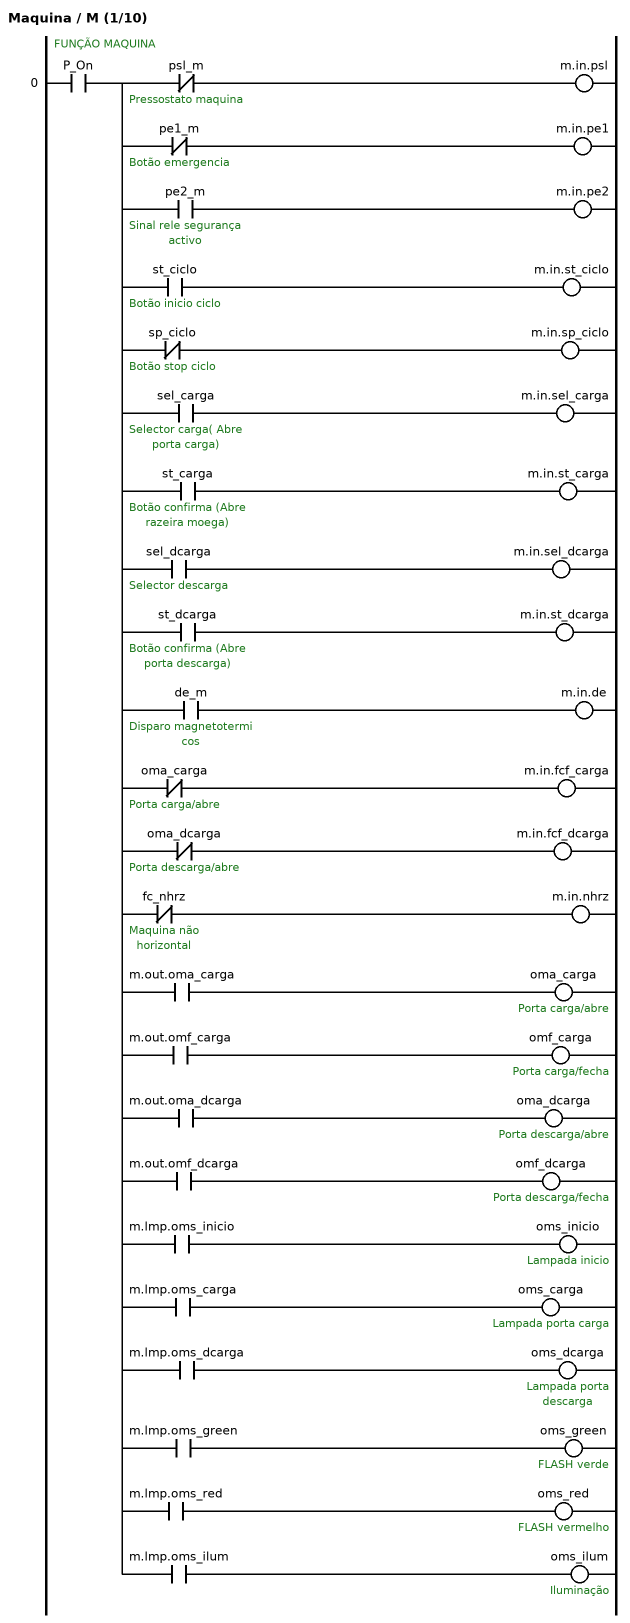
; rung 0: FUNÇÃO MAQUINA
LD P_On
OUT TR0
ANDNOT psl_m  ; Pressostato maquina
OUT m.in.psl
LD TR0
ANDNOT pe1_m  ; Botão emergencia
OUT m.in.pe1
LD TR0
AND pe2_m  ; Sinal rele segurança activo
OUT m.in.pe2
LD TR0
AND st_ciclo  ; Botão inicio ciclo
OUT m.in.st_ciclo
LD TR0
ANDNOT sp_ciclo  ; Botão stop ciclo
OUT m.in.sp_ciclo
LD TR0
AND sel_carga  ; Selector carga( Abre porta carga)
OUT m.in.sel_carga
LD TR0
AND st_carga  ; Botão confirma (Abre razeira moega)
OUT m.in.st_carga
LD TR0
AND sel_dcarga  ; Selector descarga
OUT m.in.sel_dcarga
LD TR0
AND st_dcarga  ; Botão confirma (Abre porta descarga)
OUT m.in.st_dcarga
LD TR0
AND de_m  ; Disparo magnetotermicos
OUT m.in.de
LD TR0
ANDNOT oma_carga  ; Porta carga/abre
OUT m.in.fcf_carga
LD TR0
ANDNOT oma_dcarga  ; Porta descarga/abre
OUT m.in.fcf_dcarga
LD TR0
ANDNOT fc_nhrz  ; Maquina não horizontal
OUT m.in.nhrz
LD TR0
AND m.out.oma_carga
OUT oma_carga  ; Porta carga/abre
LD TR0
AND m.out.omf_carga
OUT omf_carga  ; Porta carga/fecha
LD TR0
AND m.out.oma_dcarga
OUT oma_dcarga  ; Porta descarga/abre
LD TR0
AND m.out.omf_dcarga
OUT omf_dcarga  ; Porta descarga/fecha
LD TR0
AND m.lmp.oms_inicio
OUT oms_inicio  ; Lampada inicio
LD TR0
AND m.lmp.oms_carga
OUT oms_carga  ; Lampada porta carga
LD TR0
AND m.lmp.oms_dcarga
OUT oms_dcarga  ; Lampada porta descarga
LD TR0
AND m.lmp.oms_green
OUT oms_green  ; FLASH verde
LD TR0
AND m.lmp.oms_red
OUT oms_red  ; FLASH vermelho
LD TR0
AND m.lmp.oms_ilum
OUT oms_ilum  ; Iluminação

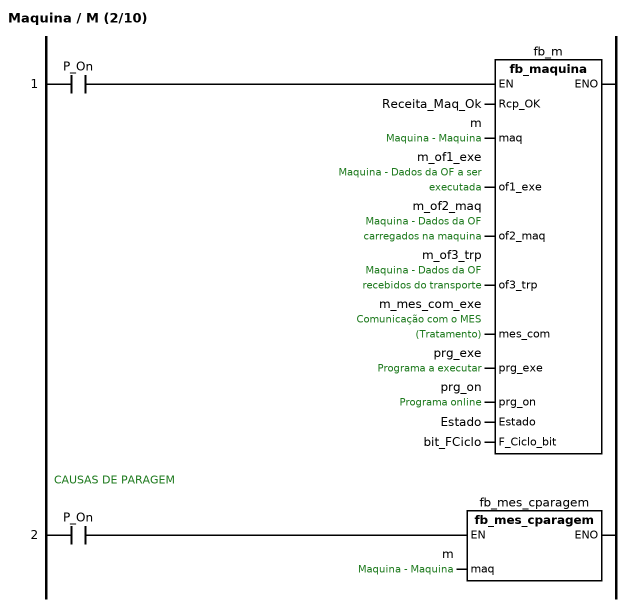
; rung 1
LD P_On
CALL fb_m : fb_maquina (Rcp_OK := Receita_Maq_Ok, maq := m, of1_exe := m_of1_exe, of2_maq := m_of2_maq, of3_trp := m_of3_trp, mes_com := m_mes_com_exe, prg_exe := prg_exe, prg_on := prg_on, Estado := Estado, F_Ciclo_bit := bit_FCiclo)  ; Maquina - Maquina, Maquina - Dados da OF a ser executada, Maquina - Dados da OF carregados na maquina, Maquina - Dados da OF recebidos do transporte, Comunicação com o MES (Tratamento), Programa a executar, Programa online
; rung 2: CAUSAS DE PARAGEM
LD P_On
CALL fb_mes_cparagem : fb_mes_cparagem (maq := m)  ; Maquina - Maquina

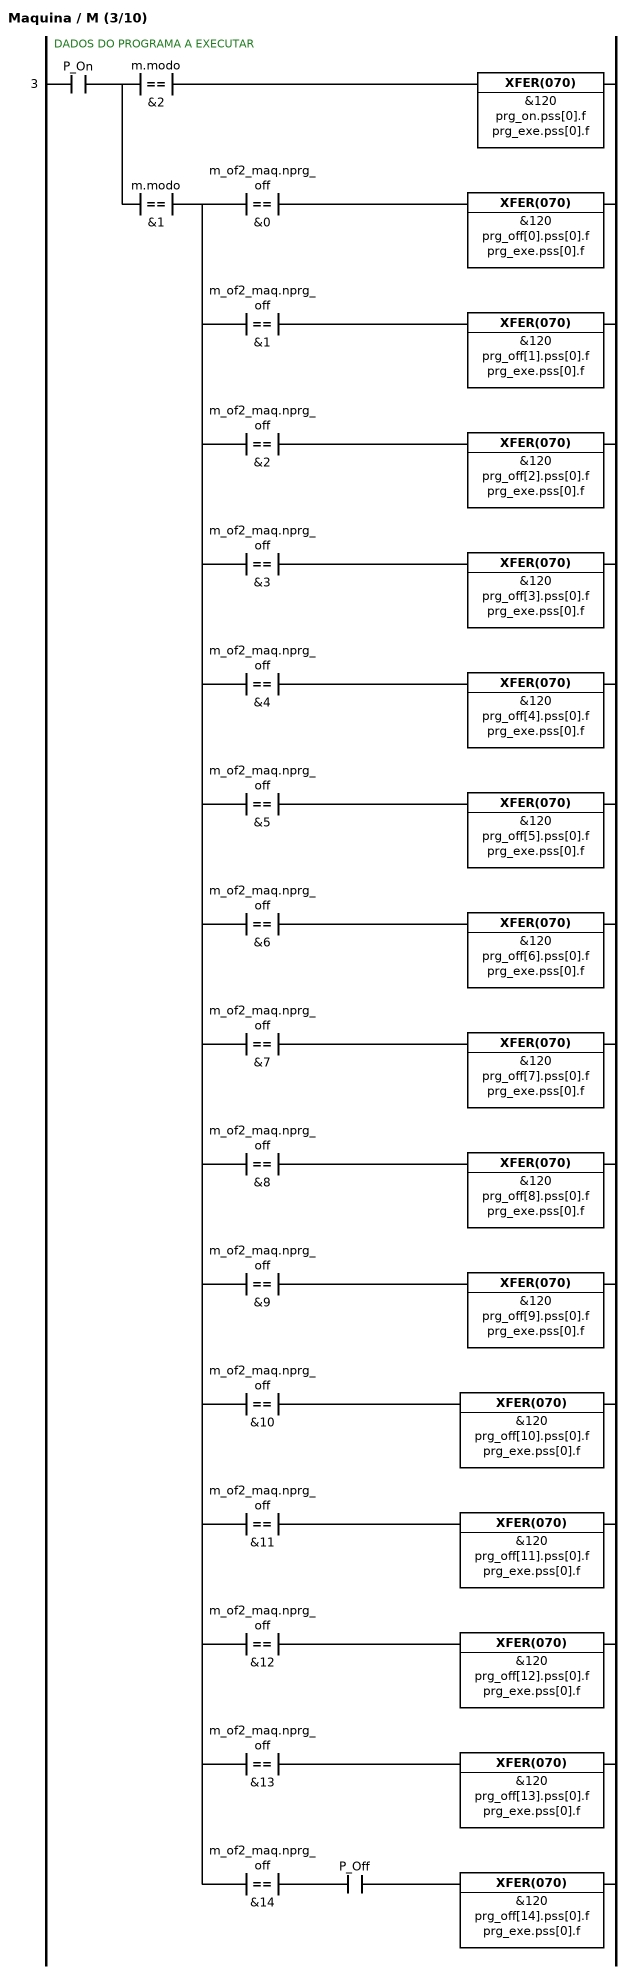
; rung 3: DADOS DO PROGRAMA A EXECUTAR
LD P_On
OUT TR0
AND=S(302) m.modo &2
XFER(070) &120 prg_on.pss[0].f prg_exe.pss[0].f
LD TR0
AND=S(302) m.modo &1
OUT TR0
AND=S(302) m_of2_maq.nprg_off &0
XFER(070) &120 prg_off[0].pss[0].f prg_exe.pss[0].f
LD TR0
AND=S(302) m_of2_maq.nprg_off &1
XFER(070) &120 prg_off[1].pss[0].f prg_exe.pss[0].f
LD TR0
AND=S(302) m_of2_maq.nprg_off &2
XFER(070) &120 prg_off[2].pss[0].f prg_exe.pss[0].f
LD TR0
AND=S(302) m_of2_maq.nprg_off &3
XFER(070) &120 prg_off[3].pss[0].f prg_exe.pss[0].f
LD TR0
AND=S(302) m_of2_maq.nprg_off &4
XFER(070) &120 prg_off[4].pss[0].f prg_exe.pss[0].f
LD TR0
AND=S(302) m_of2_maq.nprg_off &5
XFER(070) &120 prg_off[5].pss[0].f prg_exe.pss[0].f
LD TR0
AND=S(302) m_of2_maq.nprg_off &6
XFER(070) &120 prg_off[6].pss[0].f prg_exe.pss[0].f
LD TR0
AND=S(302) m_of2_maq.nprg_off &7
XFER(070) &120 prg_off[7].pss[0].f prg_exe.pss[0].f
LD TR0
AND=S(302) m_of2_maq.nprg_off &8
XFER(070) &120 prg_off[8].pss[0].f prg_exe.pss[0].f
LD TR0
AND=S(302) m_of2_maq.nprg_off &9
XFER(070) &120 prg_off[9].pss[0].f prg_exe.pss[0].f
LD TR0
AND=S(302) m_of2_maq.nprg_off &10
XFER(070) &120 prg_off[10].pss[0].f prg_exe.pss[0].f
LD TR0
AND=S(302) m_of2_maq.nprg_off &11
XFER(070) &120 prg_off[11].pss[0].f prg_exe.pss[0].f
LD TR0
AND=S(302) m_of2_maq.nprg_off &12
XFER(070) &120 prg_off[12].pss[0].f prg_exe.pss[0].f
LD TR0
AND=S(302) m_of2_maq.nprg_off &13
XFER(070) &120 prg_off[13].pss[0].f prg_exe.pss[0].f
LD TR0
AND=S(302) m_of2_maq.nprg_off &14
AND P_Off
XFER(070) &120 prg_off[14].pss[0].f prg_exe.pss[0].f

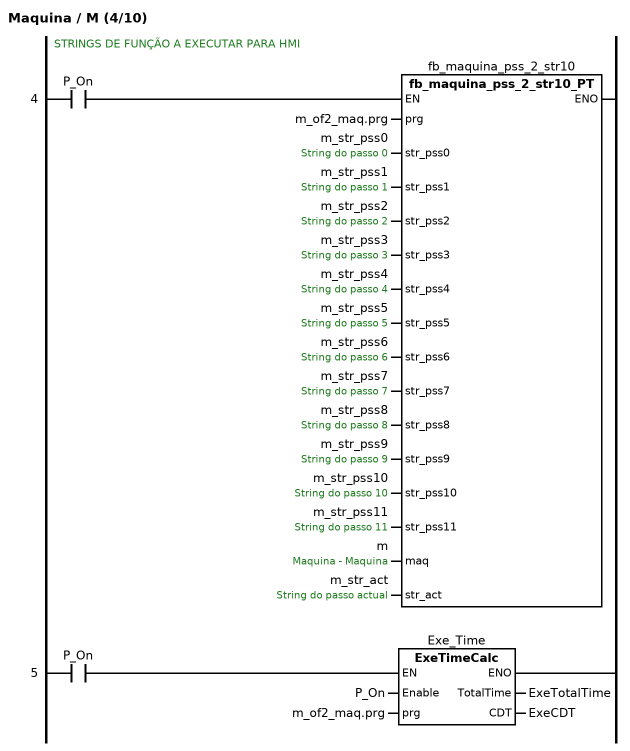
; rung 4: STRINGS DE FUNÇÃO A EXECUTAR PARA HMI
LD P_On
CALL fb_maquina_pss_2_str10 : fb_maquina_pss_2_str10_PT (prg := m_of2_maq.prg, str_pss0 := m_str_pss0, str_pss1 := m_str_pss1, str_pss2 := m_str_pss2, str_pss3 := m_str_pss3, str_pss4 := m_str_pss4, str_pss5 := m_str_pss5, str_pss6 := m_str_pss6, str_pss7 := m_str_pss7, str_pss8 := m_str_pss8, str_pss9 := m_str_pss9, str_pss10 := m_str_pss10, str_pss11 := m_str_pss11, maq := m, str_act := m_str_act)  ; String do passo 0, String do passo 1, String do passo 2, String do passo 3, String do passo 4, String do passo 5, String do passo 6, String do passo 7, String do passo 8, String do passo 9, String do passo 10, String do passo 11, Maquina - Maquina, String do passo actual
; rung 5
LD P_On
CALL Exe_Time : ExeTimeCalc (Enable := P_On, prg := m_of2_maq.prg, TotalTime => ExeTotalTime, CDT => ExeCDT)

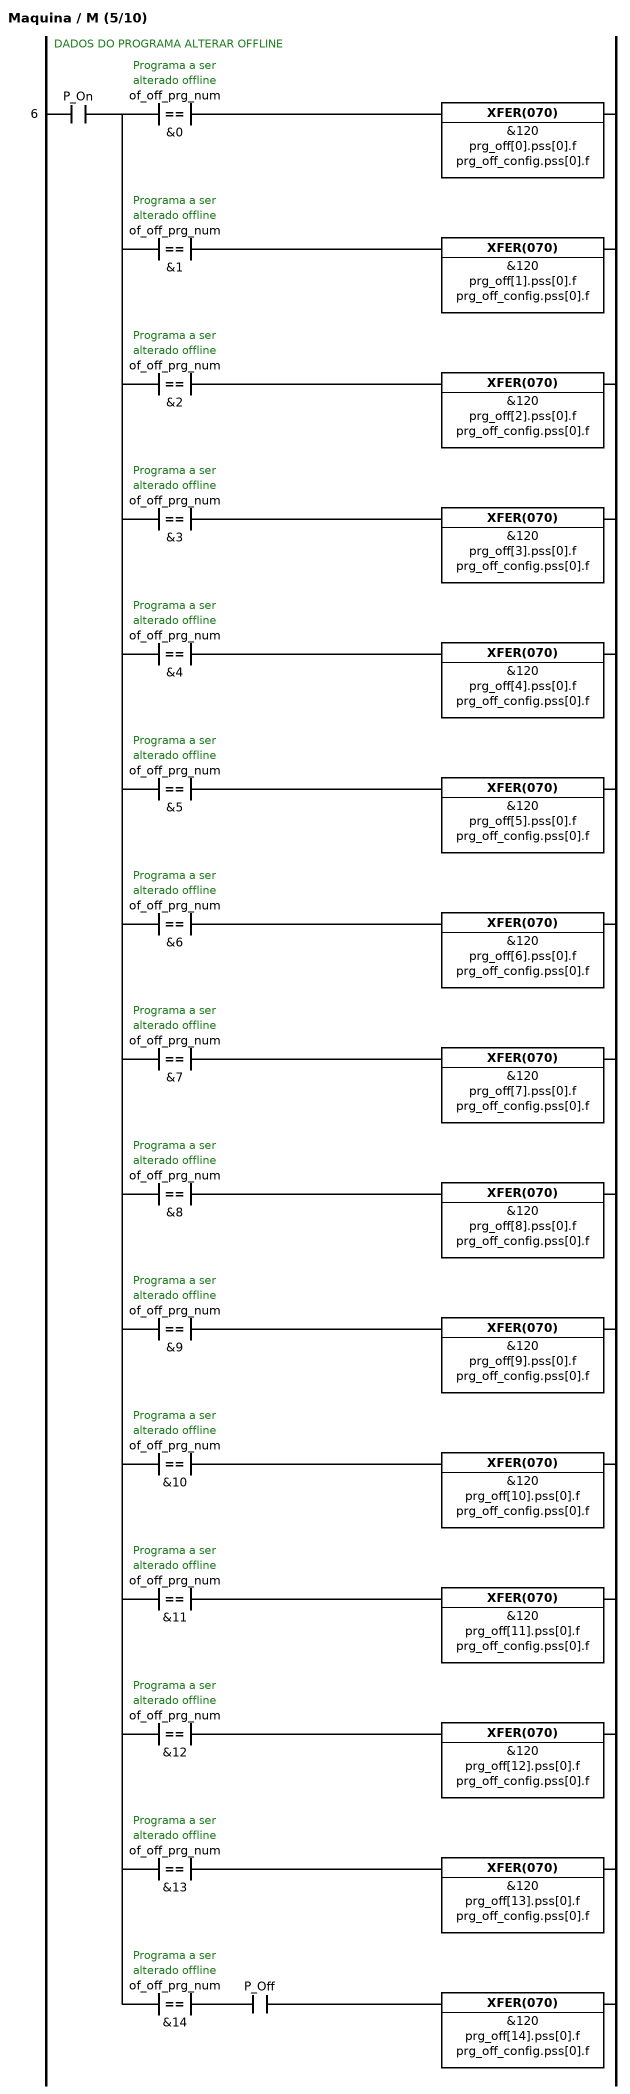
; rung 6: DADOS DO PROGRAMA ALTERAR OFFLINE
LD P_On
OUT TR0
AND=S(302) of_off_prg_num &0  ; Programa a ser alterado offline
XFER(070) &120 prg_off[0].pss[0].f prg_off_config.pss[0].f
LD TR0
AND=S(302) of_off_prg_num &1  ; Programa a ser alterado offline
XFER(070) &120 prg_off[1].pss[0].f prg_off_config.pss[0].f
LD TR0
AND=S(302) of_off_prg_num &2  ; Programa a ser alterado offline
XFER(070) &120 prg_off[2].pss[0].f prg_off_config.pss[0].f
LD TR0
AND=S(302) of_off_prg_num &3  ; Programa a ser alterado offline
XFER(070) &120 prg_off[3].pss[0].f prg_off_config.pss[0].f
LD TR0
AND=S(302) of_off_prg_num &4  ; Programa a ser alterado offline
XFER(070) &120 prg_off[4].pss[0].f prg_off_config.pss[0].f
LD TR0
AND=S(302) of_off_prg_num &5  ; Programa a ser alterado offline
XFER(070) &120 prg_off[5].pss[0].f prg_off_config.pss[0].f
LD TR0
AND=S(302) of_off_prg_num &6  ; Programa a ser alterado offline
XFER(070) &120 prg_off[6].pss[0].f prg_off_config.pss[0].f
LD TR0
AND=S(302) of_off_prg_num &7  ; Programa a ser alterado offline
XFER(070) &120 prg_off[7].pss[0].f prg_off_config.pss[0].f
LD TR0
AND=S(302) of_off_prg_num &8  ; Programa a ser alterado offline
XFER(070) &120 prg_off[8].pss[0].f prg_off_config.pss[0].f
LD TR0
AND=S(302) of_off_prg_num &9  ; Programa a ser alterado offline
XFER(070) &120 prg_off[9].pss[0].f prg_off_config.pss[0].f
LD TR0
AND=S(302) of_off_prg_num &10  ; Programa a ser alterado offline
XFER(070) &120 prg_off[10].pss[0].f prg_off_config.pss[0].f
LD TR0
AND=S(302) of_off_prg_num &11  ; Programa a ser alterado offline
XFER(070) &120 prg_off[11].pss[0].f prg_off_config.pss[0].f
LD TR0
AND=S(302) of_off_prg_num &12  ; Programa a ser alterado offline
XFER(070) &120 prg_off[12].pss[0].f prg_off_config.pss[0].f
LD TR0
AND=S(302) of_off_prg_num &13  ; Programa a ser alterado offline
XFER(070) &120 prg_off[13].pss[0].f prg_off_config.pss[0].f
LD TR0
AND=S(302) of_off_prg_num &14  ; Programa a ser alterado offline
AND P_Off
XFER(070) &120 prg_off[14].pss[0].f prg_off_config.pss[0].f

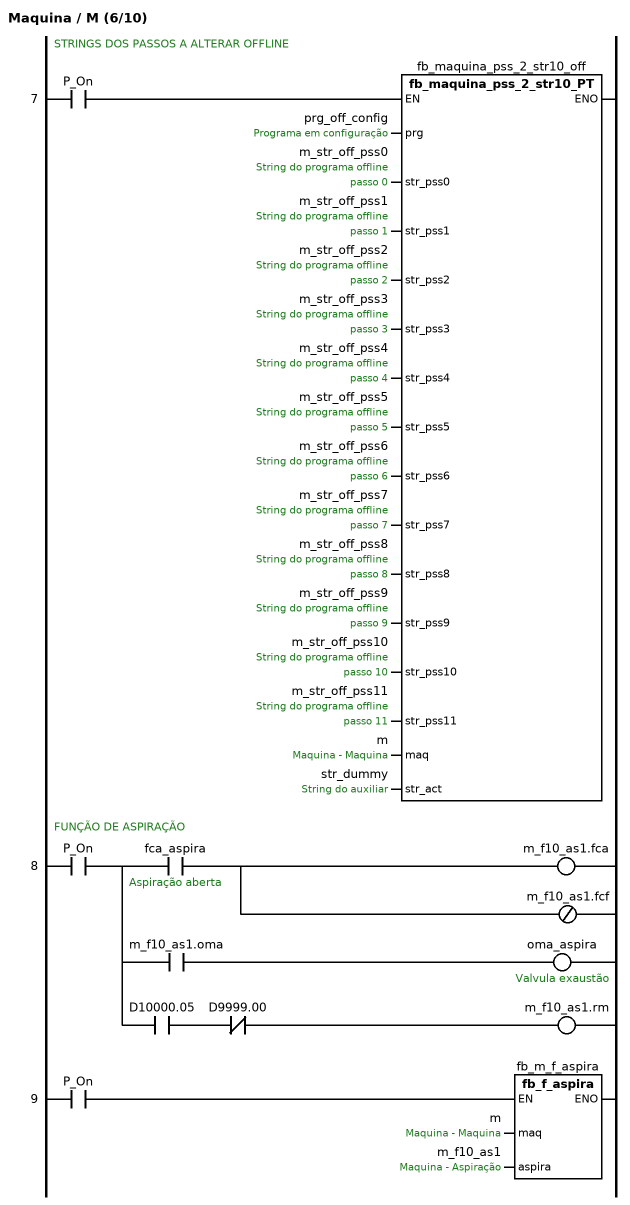
; rung 7: STRINGS DOS PASSOS A ALTERAR OFFLINE
LD P_On
CALL fb_maquina_pss_2_str10_off : fb_maquina_pss_2_str10_PT (prg := prg_off_config, str_pss0 := m_str_off_pss0, str_pss1 := m_str_off_pss1, str_pss2 := m_str_off_pss2, str_pss3 := m_str_off_pss3, str_pss4 := m_str_off_pss4, str_pss5 := m_str_off_pss5, str_pss6 := m_str_off_pss6, str_pss7 := m_str_off_pss7, str_pss8 := m_str_off_pss8, str_pss9 := m_str_off_pss9, str_pss10 := m_str_off_pss10, str_pss11 := m_str_off_pss11, maq := m, str_act := str_dummy)  ; Programa em configuração, String do programa offline passo 0, String do programa offline passo 1, String do programa offline passo 2, String do programa offline passo 3, String do programa offline passo 4, String do programa offline passo 5, String do programa offline passo 6, String do programa offline passo 7, String do programa offline passo 8, String do programa offline passo 9, String do programa offline passo 10, String do programa offline passo 11, Maquina - Maquina, String do auxiliar
; rung 8: FUNÇÃO DE ASPIRAÇÃO
LD P_On
OUT TR0
AND fca_aspira  ; Aspiração aberta
OUT m_f10_as1.fca
OUTNOT m_f10_as1.fcf
LD TR0
AND m_f10_as1.oma
OUT oma_aspira  ; Valvula exaustão
LD TR0
AND D10000.05
ANDNOT D9999.00
OUT m_f10_as1.rm
; rung 9
LD P_On
CALL fb_m_f_aspira : fb_f_aspira (maq := m, aspira := m_f10_as1)  ; Maquina - Maquina, Maquina - Aspiração

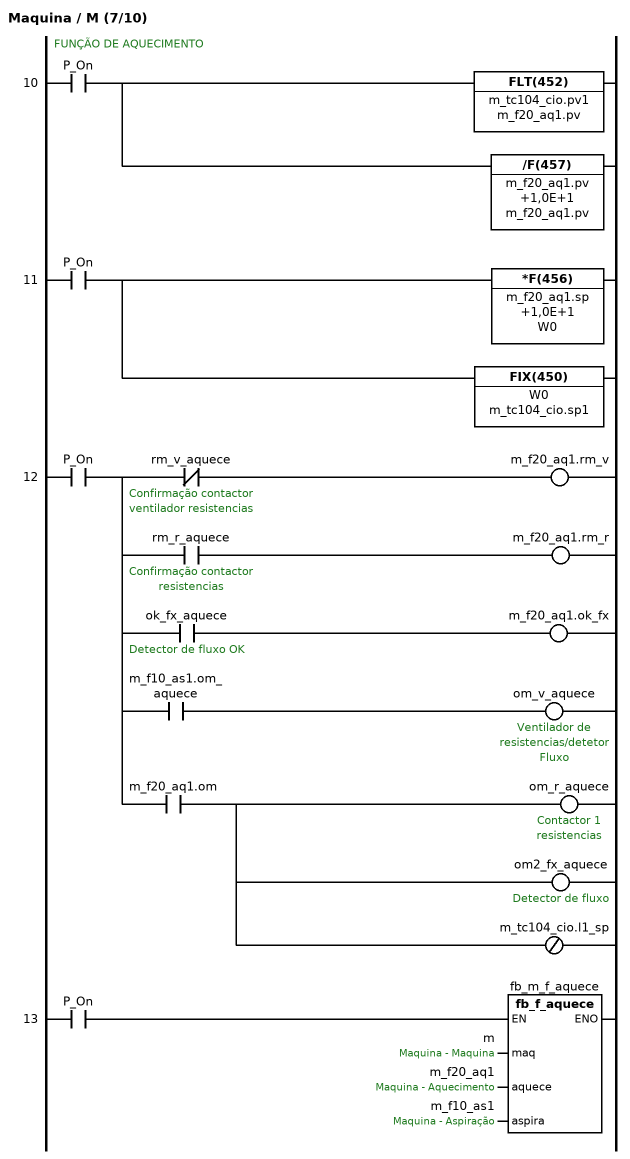
; rung 10: FUNÇÃO DE AQUECIMENTO
LD P_On
FLT(452) m_tc104_cio.pv1 m_f20_aq1.pv
/F(457) m_f20_aq1.pv +1,0E+1 m_f20_aq1.pv
; rung 11
LD P_On
*F(456) m_f20_aq1.sp +1,0E+1 W0
FIX(450) W0 m_tc104_cio.sp1
; rung 12
LD P_On
OUT TR0
ANDNOT rm_v_aquece  ; Confirmação contactor ventilador resistencias
OUT m_f20_aq1.rm_v
LD TR0
AND rm_r_aquece  ; Confirmação contactor resistencias
OUT m_f20_aq1.rm_r
LD TR0
AND ok_fx_aquece  ; Detector de fluxo OK
OUT m_f20_aq1.ok_fx
LD TR0
AND m_f10_as1.om_aquece
OUT om_v_aquece  ; Ventilador de resistencias/detetor Fluxo
LD TR0
AND m_f20_aq1.om
OUT om_r_aquece  ; Contactor 1 resistencias
OUT om2_fx_aquece  ; Detector de fluxo
OUTNOT m_tc104_cio.l1_sp
; rung 13
LD P_On
CALL fb_m_f_aquece : fb_f_aquece (maq := m, aquece := m_f20_aq1, aspira := m_f10_as1)  ; Maquina - Maquina, Maquina - Aquecimento, Maquina - Aspiração

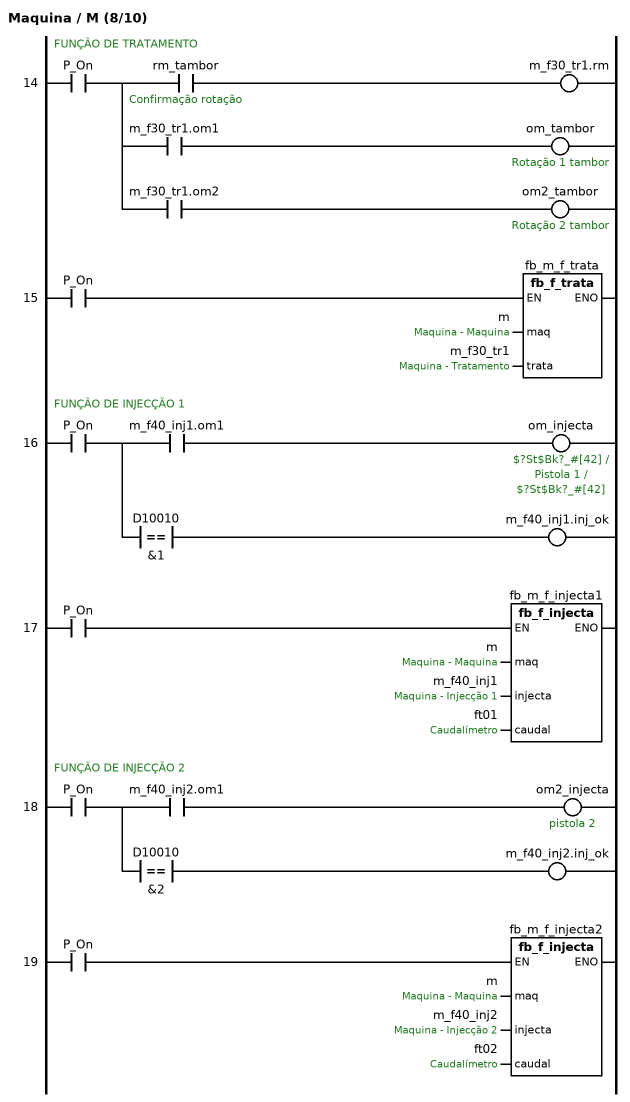
; rung 14: FUNÇÃO DE TRATAMENTO
LD P_On
OUT TR0
AND rm_tambor  ; Confirmação rotação
OUT m_f30_tr1.rm
LD TR0
AND m_f30_tr1.om1
OUT om_tambor  ; Rotação 1 tambor
LD TR0
AND m_f30_tr1.om2
OUT om2_tambor  ; Rotação 2 tambor
; rung 15
LD P_On
CALL fb_m_f_trata : fb_f_trata (maq := m, trata := m_f30_tr1)  ; Maquina - Maquina, Maquina - Tratamento
; rung 16: FUNÇÃO DE INJECÇÃO 1
LD P_On
OUT TR0
AND m_f40_inj1.om1
OUT om_injecta  ; $?St$Bk?_#[42] / Pistola 1 / $?St$Bk?_#[42]
LD TR0
AND=(300) D10010 &1
OUT m_f40_inj1.inj_ok
; rung 17
LD P_On
CALL fb_m_f_injecta1 : fb_f_injecta (maq := m, injecta := m_f40_inj1, caudal := ft01)  ; Maquina - Maquina, Maquina - Injecção 1, Caudalímetro
; rung 18: FUNÇÃO DE INJECÇÃO 2
LD P_On
OUT TR0
AND m_f40_inj2.om1
OUT om2_injecta  ; pistola 2
LD TR0
AND=(300) D10010 &2
OUT m_f40_inj2.inj_ok
; rung 19
LD P_On
CALL fb_m_f_injecta2 : fb_f_injecta (maq := m, injecta := m_f40_inj2, caudal := ft02)  ; Maquina - Maquina, Maquina - Injecção 2, Caudalímetro

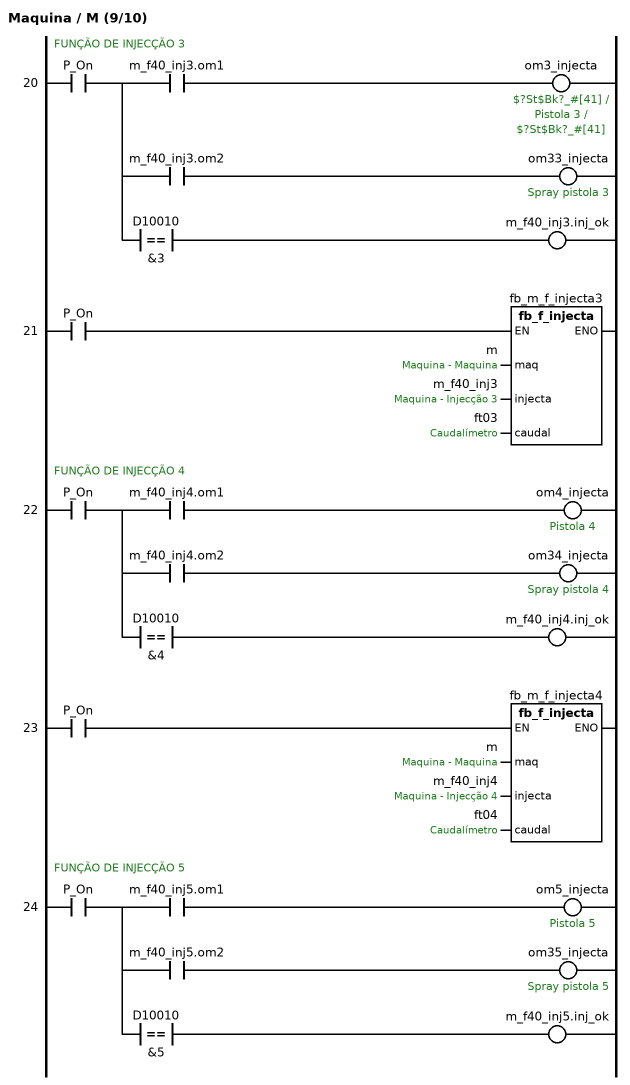
; rung 20: FUNÇÃO DE INJECÇÃO 3
LD P_On
OUT TR0
AND m_f40_inj3.om1
OUT om3_injecta  ; $?St$Bk?_#[41] / Pistola 3 / $?St$Bk?_#[41]
LD TR0
AND m_f40_inj3.om2
OUT om33_injecta  ; Spray pistola 3
LD TR0
AND=(300) D10010 &3
OUT m_f40_inj3.inj_ok
; rung 21
LD P_On
CALL fb_m_f_injecta3 : fb_f_injecta (maq := m, injecta := m_f40_inj3, caudal := ft03)  ; Maquina - Maquina, Maquina - Injecção 3, Caudalímetro
; rung 22: FUNÇÃO DE INJECÇÃO 4
LD P_On
OUT TR0
AND m_f40_inj4.om1
OUT om4_injecta  ; Pistola 4
LD TR0
AND m_f40_inj4.om2
OUT om34_injecta  ; Spray pistola 4
LD TR0
AND=(300) D10010 &4
OUT m_f40_inj4.inj_ok
; rung 23
LD P_On
CALL fb_m_f_injecta4 : fb_f_injecta (maq := m, injecta := m_f40_inj4, caudal := ft04)  ; Maquina - Maquina, Maquina - Injecção 4, Caudalímetro
; rung 24: FUNÇÃO DE INJECÇÃO 5
LD P_On
OUT TR0
AND m_f40_inj5.om1
OUT om5_injecta  ; Pistola 5
LD TR0
AND m_f40_inj5.om2
OUT om35_injecta  ; Spray pistola 5
LD TR0
AND=(300) D10010 &5
OUT m_f40_inj5.inj_ok

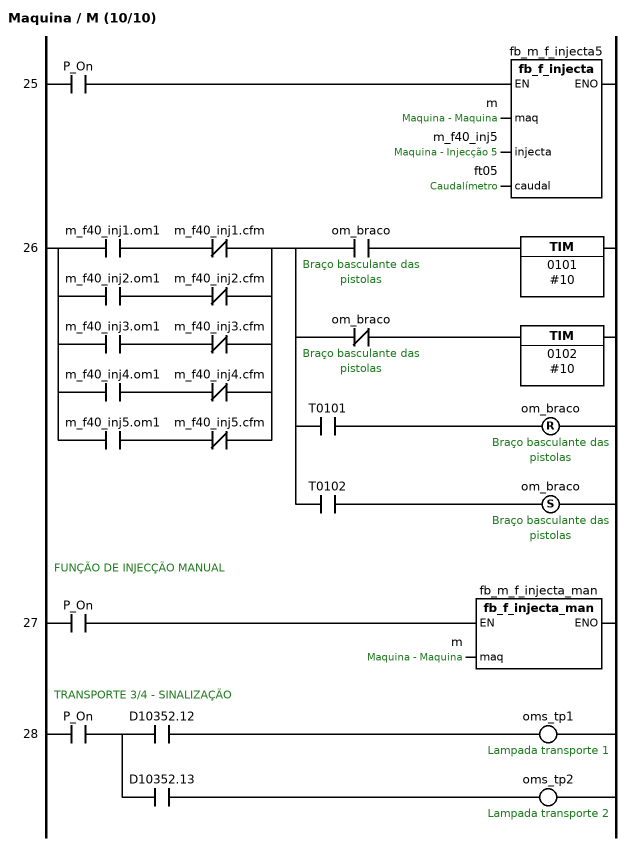
; rung 25
LD P_On
CALL fb_m_f_injecta5 : fb_f_injecta (maq := m, injecta := m_f40_inj5, caudal := ft05)  ; Maquina - Maquina, Maquina - Injecção 5, Caudalímetro
; rung 26
LD m_f40_inj1.om1
ANDNOT m_f40_inj1.cfm
LD m_f40_inj2.om1
ANDNOT m_f40_inj2.cfm
ORLD
LD m_f40_inj3.om1
ANDNOT m_f40_inj3.cfm
ORLD
LD m_f40_inj4.om1
ANDNOT m_f40_inj4.cfm
ORLD
LD m_f40_inj5.om1
ANDNOT m_f40_inj5.cfm
ORLD
OUT TR0
AND om_braco  ; Braço basculante das pistolas
TIM 0101 #10
LD TR0
ANDNOT om_braco  ; Braço basculante das pistolas
TIM 0102 #10
LD TR0
AND T0101
RSET om_braco  ; Braço basculante das pistolas
LD TR0
AND T0102
SET om_braco  ; Braço basculante das pistolas
; rung 27: FUNÇÃO DE INJECÇÃO MANUAL
LD P_On
CALL fb_m_f_injecta_man : fb_f_injecta_man (maq := m)  ; Maquina - Maquina
; rung 28: TRANSPORTE 3/4 - SINALIZAÇÃO
LD P_On
OUT TR0
AND D10352.12
OUT oms_tp1  ; Lampada transporte 1
LD TR0
AND D10352.13
OUT oms_tp2  ; Lampada transporte 2

### Section New_MES

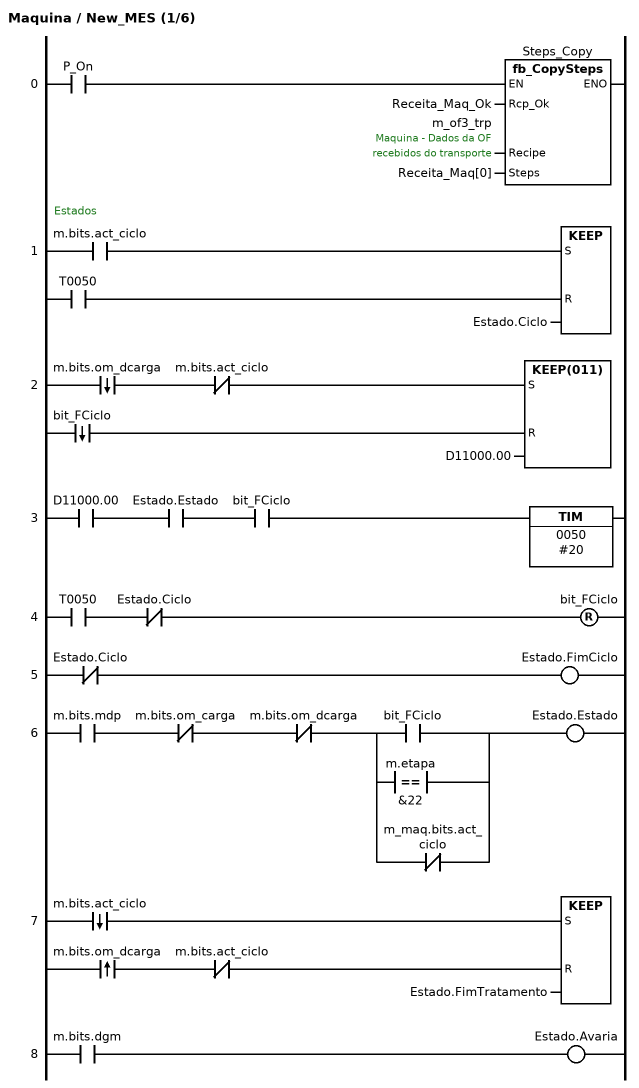
; rung 0
LD P_On
CALL Steps_Copy : fb_CopySteps (Rcp_Ok := Receita_Maq_Ok, Recipe := m_of3_trp, Steps := Receita_Maq[0])  ; Maquina - Dados da OF recebidos do transporte
; rung 1: Estados
LD m.bits.act_ciclo
LD T0050
KEEP Estado.Ciclo
; rung 2
%LD m.bits.om_dcarga
ANDNOT m.bits.act_ciclo
%LD bit_FCiclo
KEEP(011) D11000.00
; rung 3
LD D11000.00
AND Estado.Estado
AND bit_FCiclo
TIM 0050 #20
; rung 4
LD T0050
ANDNOT Estado.Ciclo
RSET bit_FCiclo
; rung 5
LDNOT Estado.Ciclo
OUT Estado.FimCiclo
; rung 6
LD m.bits.mdp
ANDNOT m.bits.om_carga
ANDNOT m.bits.om_dcarga
LD bit_FCiclo
OR=(300) m.etapa &22
ORNOT m_maq.bits.act_ciclo
ANDLD
OUT Estado.Estado
; rung 7
%LD m.bits.act_ciclo
@LD m.bits.om_dcarga
ANDNOT m.bits.act_ciclo
KEEP Estado.FimTratamento
; rung 8
LD m.bits.dgm
OUT Estado.Avaria

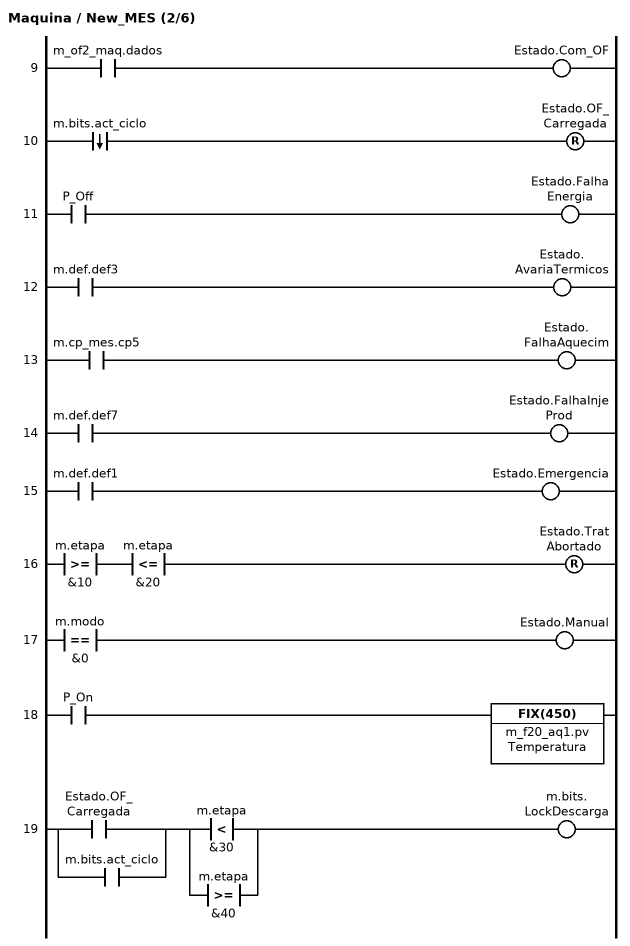
; rung 9
LD m_of2_maq.dados
OUT Estado.Com_OF
; rung 10
%LD m.bits.act_ciclo
RSET Estado.OF_Carregada
; rung 11
LD P_Off
OUT Estado.FalhaEnergia
; rung 12
LD m.def.def3
OUT Estado.AvariaTermicos
; rung 13
LD m.cp_mes.cp5
OUT Estado.FalhaAquecim
; rung 14
LD m.def.def7
OUT Estado.FalhaInjeProd
; rung 15
LD m.def.def1
OUT Estado.Emergencia
; rung 16
LD>=S(327) m.etapa &10
AND<=S(317) m.etapa &20
RSET Estado.TratAbortado
; rung 17
LD=(300) m.modo &0
OUT Estado.Manual
; rung 18
LD P_On
FIX(450) m_f20_aq1.pv Temperatura
; rung 19
LD Estado.OF_Carregada
OR m.bits.act_ciclo
LD<(310) m.etapa &30
OR>=(325) m.etapa &40
ANDLD
OUT m.bits.LockDescarga

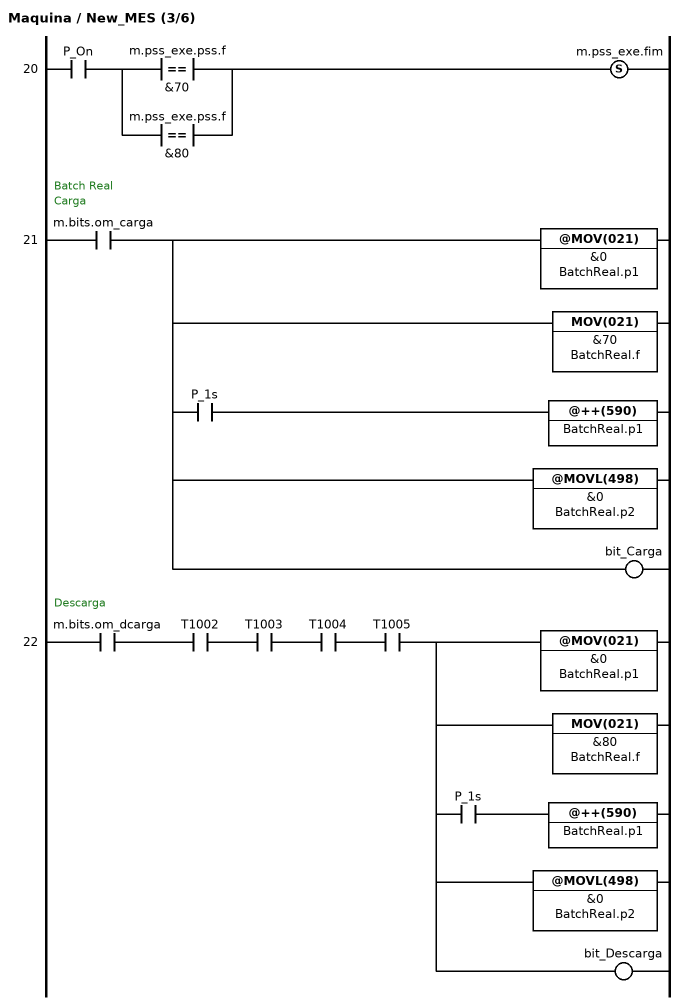
; rung 20
LD P_On
LD=(300) m.pss_exe.pss.f &70
OR=(300) m.pss_exe.pss.f &80
ANDLD
SET m.pss_exe.fim
; rung 21: Batch Real / Carga
LD m.bits.om_carga
OUT TR0
@MOV(021) &0 BatchReal.p1
MOV(021) &70 BatchReal.f
AND P_1s
@++(590) BatchReal.p1
LD TR0
@MOVL(498) &0 BatchReal.p2
OUT bit_Carga
; rung 22: Descarga
LD m.bits.om_dcarga
AND T1002
AND T1003
AND T1004
AND T1005
OUT TR0
@MOV(021) &0 BatchReal.p1
MOV(021) &80 BatchReal.f
AND P_1s
@++(590) BatchReal.p1
LD TR0
@MOVL(498) &0 BatchReal.p2
OUT bit_Descarga

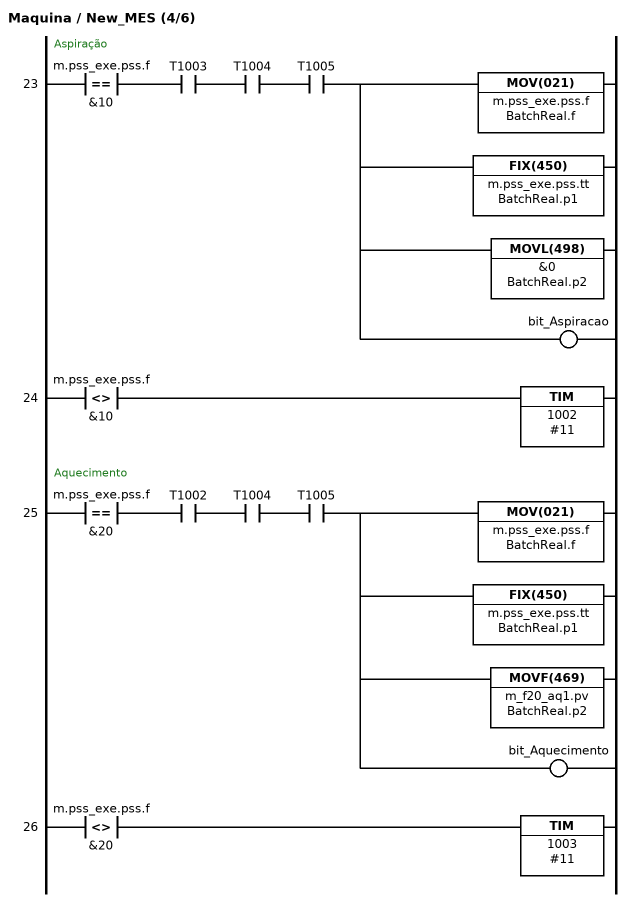
; rung 23: Aspiração
LD=(300) m.pss_exe.pss.f &10
AND T1003
AND T1004
AND T1005
MOV(021) m.pss_exe.pss.f BatchReal.f
FIX(450) m.pss_exe.pss.tt BatchReal.p1
MOVL(498) &0 BatchReal.p2
OUT bit_Aspiracao
; rung 24
LD<>(305) m.pss_exe.pss.f &10
TIM 1002 #11
; rung 25: Aquecimento
LD=(300) m.pss_exe.pss.f &20
AND T1002
AND T1004
AND T1005
MOV(021) m.pss_exe.pss.f BatchReal.f
FIX(450) m.pss_exe.pss.tt BatchReal.p1
MOVF(469) m_f20_aq1.pv BatchReal.p2
OUT bit_Aquecimento
; rung 26
LD<>(305) m.pss_exe.pss.f &20
TIM 1003 #11

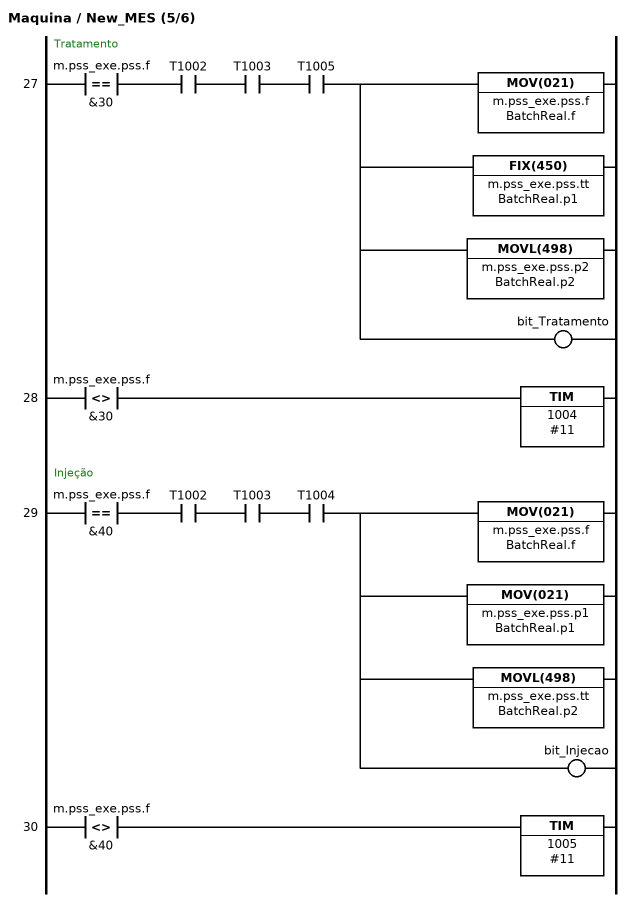
; rung 27: Tratamento
LD=(300) m.pss_exe.pss.f &30
AND T1002
AND T1003
AND T1005
MOV(021) m.pss_exe.pss.f BatchReal.f
FIX(450) m.pss_exe.pss.tt BatchReal.p1
MOVL(498) m.pss_exe.pss.p2 BatchReal.p2
OUT bit_Tratamento
; rung 28
LD<>(305) m.pss_exe.pss.f &30
TIM 1004 #11
; rung 29: Injeção
LD=(300) m.pss_exe.pss.f &40
AND T1002
AND T1003
AND T1004
MOV(021) m.pss_exe.pss.f BatchReal.f
MOV(021) m.pss_exe.pss.p1 BatchReal.p1
MOVL(498) m.pss_exe.pss.tt BatchReal.p2
OUT bit_Injecao
; rung 30
LD<>(305) m.pss_exe.pss.f &40
TIM 1005 #11

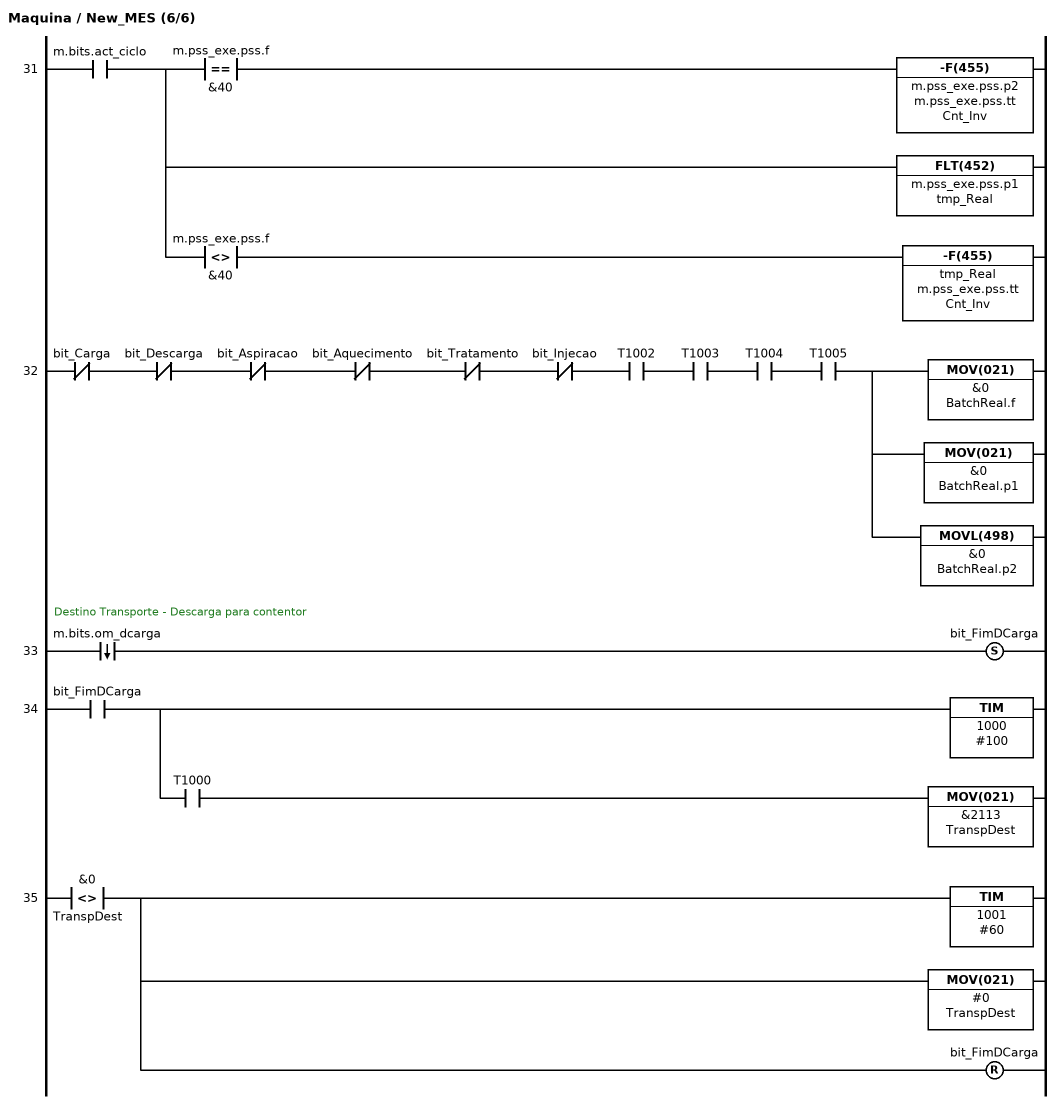
; rung 31
LD m.bits.act_ciclo
OUT TR0
AND=(300) m.pss_exe.pss.f &40
-F(455) m.pss_exe.pss.p2 m.pss_exe.pss.tt Cnt_Inv
LD TR0
FLT(452) m.pss_exe.pss.p1 tmp_Real
AND<>(305) m.pss_exe.pss.f &40
-F(455) tmp_Real m.pss_exe.pss.tt Cnt_Inv
; rung 32
LDNOT bit_Carga
ANDNOT bit_Descarga
ANDNOT bit_Aspiracao
ANDNOT bit_Aquecimento
ANDNOT bit_Tratamento
ANDNOT bit_Injecao
AND T1002
AND T1003
AND T1004
AND T1005
MOV(021) &0 BatchReal.f
MOV(021) &0 BatchReal.p1
MOVL(498) &0 BatchReal.p2
; rung 33: Destino Transporte - Descarga para contentor
%LD m.bits.om_dcarga
SET bit_FimDCarga
; rung 34
LD bit_FimDCarga
TIM 1000 #100
AND T1000
MOV(021) &2113 TranspDest
; rung 35
LD<>(305) &0 TranspDest
TIM 1001 #60
MOV(021) #0 TranspDest
RSET bit_FimDCarga

### Section M_MES
; rung 0

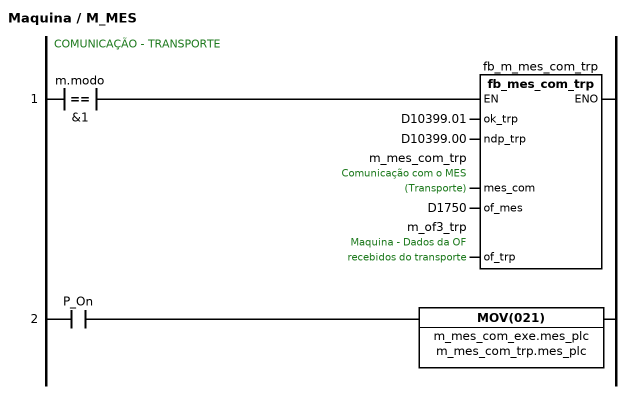
; rung 1: COMUNICAÇÃO - TRANSPORTE
LD=(300) m.modo &1
CALL fb_m_mes_com_trp : fb_mes_com_trp (ok_trp := D10399.01, ndp_trp := D10399.00, mes_com := m_mes_com_trp, of_mes := D1750, of_trp := m_of3_trp)  ; Comunicação com o MES (Transporte), Maquina - Dados da OF recebidos do transporte
; rung 2
LD P_On
MOV(021) m_mes_com_exe.mes_plc m_mes_com_trp.mes_plc

### Section FCOMUNICACAO

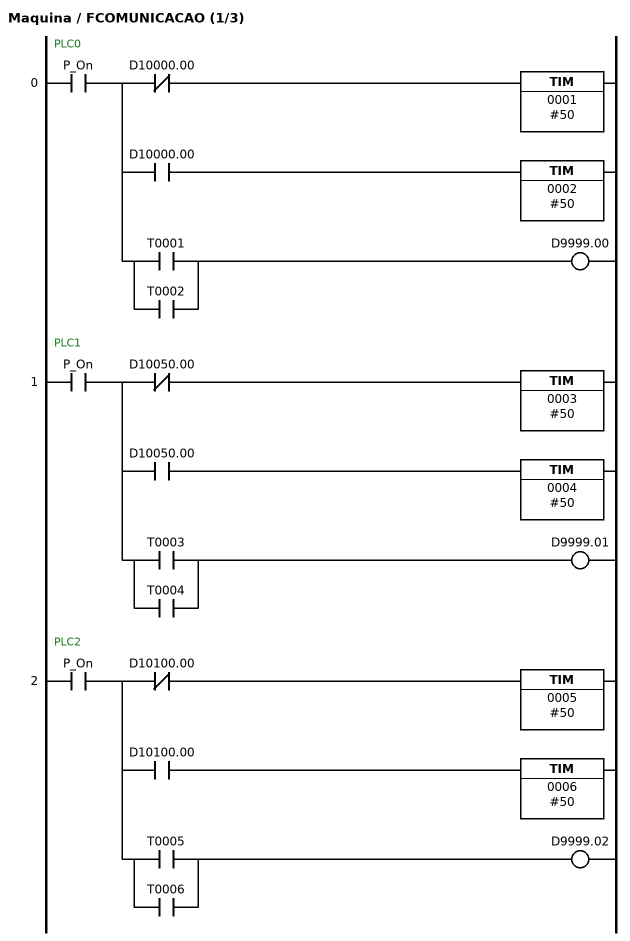
; rung 0: PLC0
LD P_On
OUT TR0
ANDNOT D10000.00
TIM 0001 #50
LD TR0
AND D10000.00
TIM 0002 #50
LD TR0
LD T0001
OR T0002
ANDLD
OUT D9999.00
; rung 1: PLC1
LD P_On
OUT TR0
ANDNOT D10050.00
TIM 0003 #50
LD TR0
AND D10050.00
TIM 0004 #50
LD TR0
LD T0003
OR T0004
ANDLD
OUT D9999.01
; rung 2: PLC2
LD P_On
OUT TR0
ANDNOT D10100.00
TIM 0005 #50
LD TR0
AND D10100.00
TIM 0006 #50
LD TR0
LD T0005
OR T0006
ANDLD
OUT D9999.02

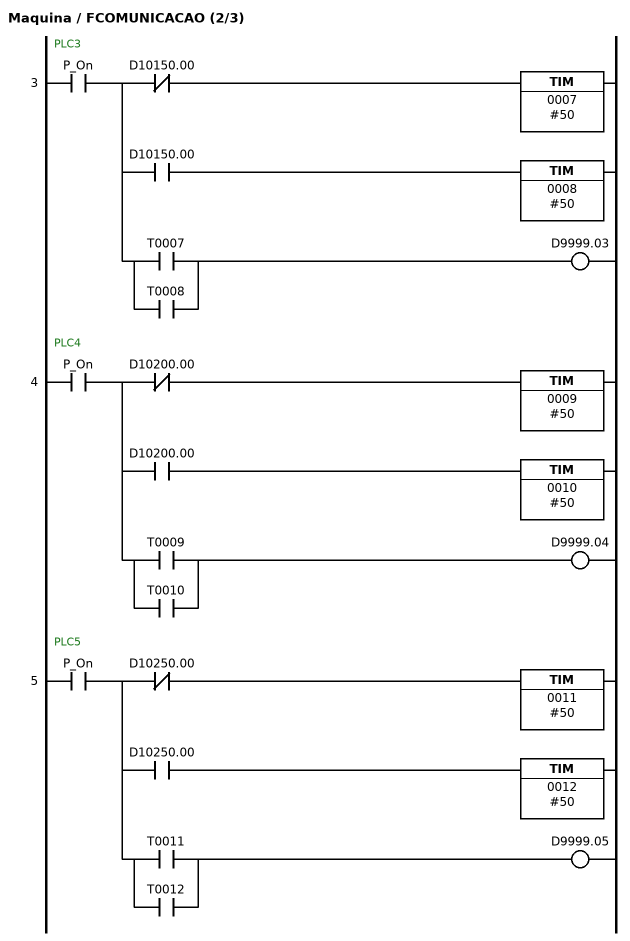
; rung 3: PLC3
LD P_On
OUT TR0
ANDNOT D10150.00
TIM 0007 #50
LD TR0
AND D10150.00
TIM 0008 #50
LD TR0
LD T0007
OR T0008
ANDLD
OUT D9999.03
; rung 4: PLC4
LD P_On
OUT TR0
ANDNOT D10200.00
TIM 0009 #50
LD TR0
AND D10200.00
TIM 0010 #50
LD TR0
LD T0009
OR T0010
ANDLD
OUT D9999.04
; rung 5: PLC5
LD P_On
OUT TR0
ANDNOT D10250.00
TIM 0011 #50
LD TR0
AND D10250.00
TIM 0012 #50
LD TR0
LD T0011
OR T0012
ANDLD
OUT D9999.05

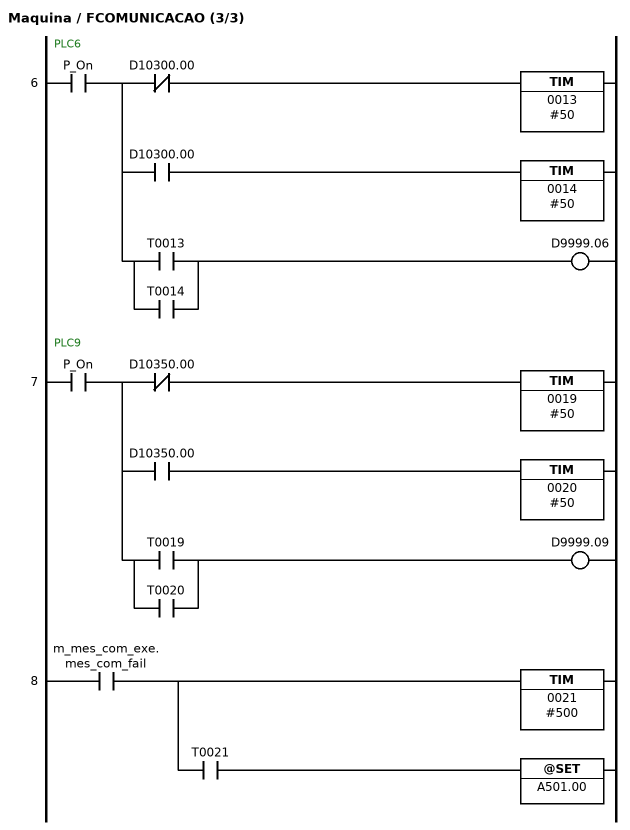
; rung 6: PLC6
LD P_On
OUT TR0
ANDNOT D10300.00
TIM 0013 #50
LD TR0
AND D10300.00
TIM 0014 #50
LD TR0
LD T0013
OR T0014
ANDLD
OUT D9999.06
; rung 7: PLC9
LD P_On
OUT TR0
ANDNOT D10350.00
TIM 0019 #50
LD TR0
AND D10350.00
TIM 0020 #50
LD TR0
LD T0019
OR T0020
ANDLD
OUT D9999.09
; rung 8
LD m_mes_com_exe.mes_com_fail
TIM 0021 #500
AND T0021
@SET A501.00

### Section COMUNICACAO

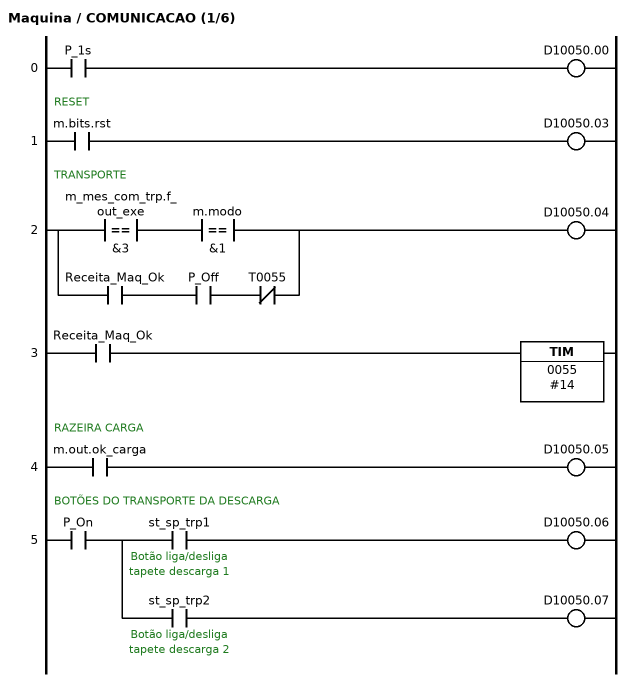
; rung 0
LD P_1s
OUT D10050.00
; rung 1: RESET
LD m.bits.rst
OUT D10050.03
; rung 2: TRANSPORTE
LD=(300) m_mes_com_trp.f_out_exe &3
AND=(300) m.modo &1
LD Receita_Maq_Ok
AND P_Off
ANDNOT T0055
ORLD
OUT D10050.04
; rung 3
LD Receita_Maq_Ok
TIM 0055 #14
; rung 4: RAZEIRA CARGA
LD m.out.ok_carga
OUT D10050.05
; rung 5: BOTÕES DO TRANSPORTE DA DESCARGA
LD P_On
OUT TR0
AND st_sp_trp1  ; Botão liga/desliga tapete descarga 1
OUT D10050.06
LD TR0
AND st_sp_trp2  ; Botão liga/desliga tapete descarga 2
OUT D10050.07

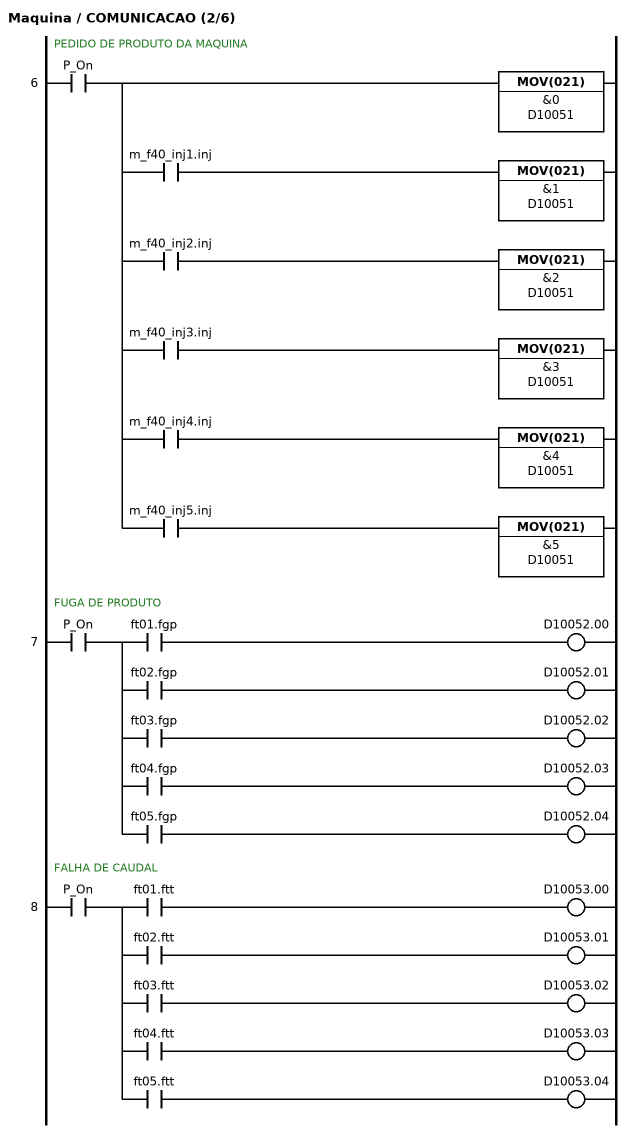
; rung 6: PEDIDO DE PRODUTO DA MAQUINA
LD P_On
OUT TR0
MOV(021) &0 D10051
AND m_f40_inj1.inj
MOV(021) &1 D10051
LD TR0
AND m_f40_inj2.inj
MOV(021) &2 D10051
LD TR0
AND m_f40_inj3.inj
MOV(021) &3 D10051
LD TR0
AND m_f40_inj4.inj
MOV(021) &4 D10051
LD TR0
AND m_f40_inj5.inj
MOV(021) &5 D10051
; rung 7: FUGA DE PRODUTO
LD P_On
OUT TR0
AND ft01.fgp
OUT D10052.00
LD TR0
AND ft02.fgp
OUT D10052.01
LD TR0
AND ft03.fgp
OUT D10052.02
LD TR0
AND ft04.fgp
OUT D10052.03
LD TR0
AND ft05.fgp
OUT D10052.04
; rung 8: FALHA DE CAUDAL
LD P_On
OUT TR0
AND ft01.ftt
OUT D10053.00
LD TR0
AND ft02.ftt
OUT D10053.01
LD TR0
AND ft03.ftt
OUT D10053.02
LD TR0
AND ft04.ftt
OUT D10053.03
LD TR0
AND ft05.ftt
OUT D10053.04

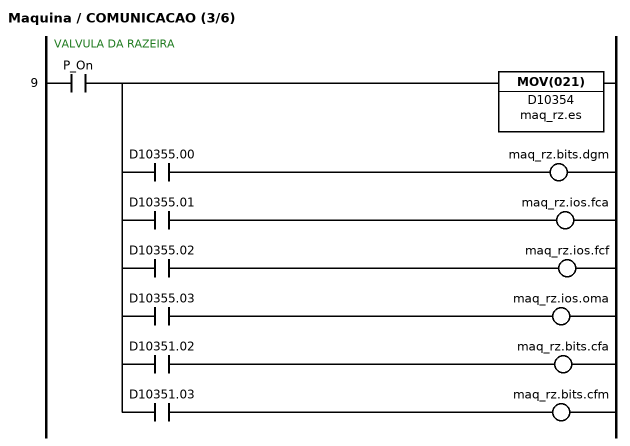
; rung 9: VALVULA DA RAZEIRA
LD P_On
OUT TR0
MOV(021) D10354 maq_rz.es
AND D10355.00
OUT maq_rz.bits.dgm
LD TR0
AND D10355.01
OUT maq_rz.ios.fca
LD TR0
AND D10355.02
OUT maq_rz.ios.fcf
LD TR0
AND D10355.03
OUT maq_rz.ios.oma
LD TR0
AND D10351.02
OUT maq_rz.bits.cfa
LD TR0
AND D10351.03
OUT maq_rz.bits.cfm

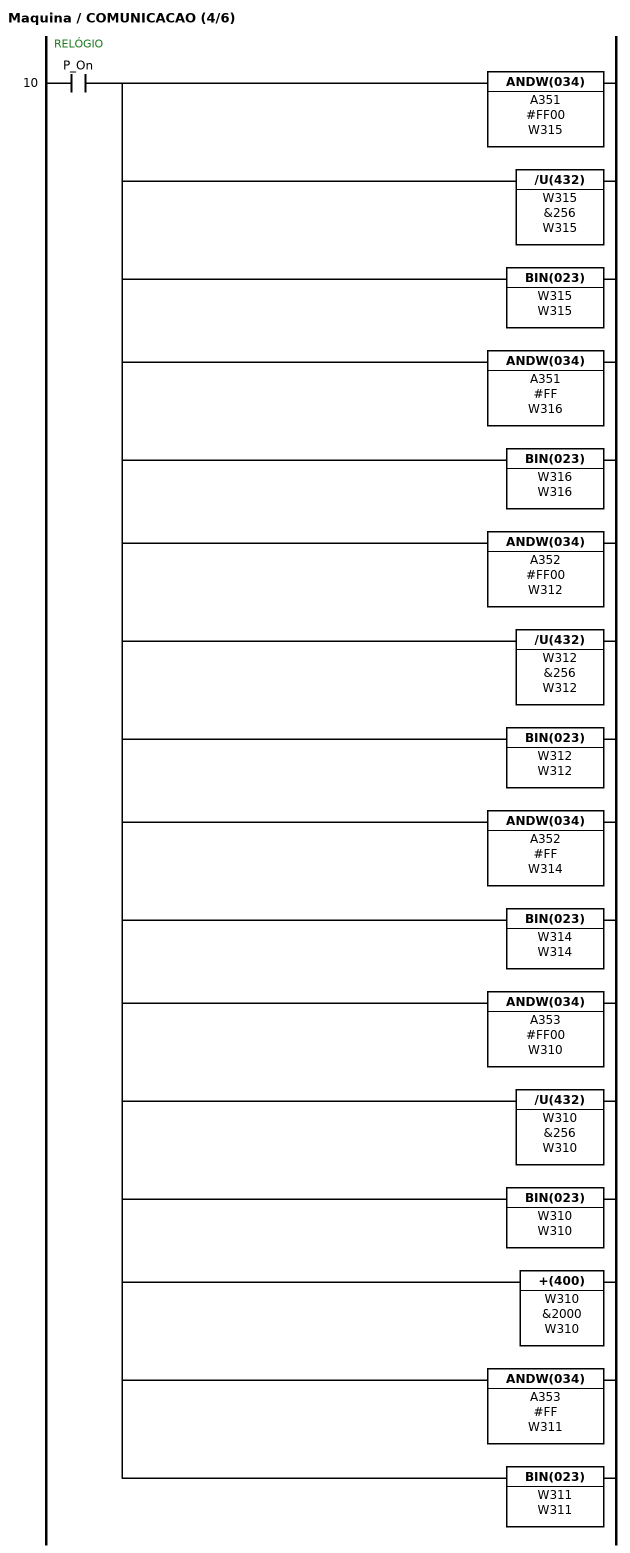
; rung 10: RELÓGIO
LD P_On
ANDW(034) A351 #FF00 W315
/U(432) W315 &256 W315
BIN(023) W315 W315
ANDW(034) A351 #FF W316
BIN(023) W316 W316
ANDW(034) A352 #FF00 W312
/U(432) W312 &256 W312
BIN(023) W312 W312
ANDW(034) A352 #FF W314
BIN(023) W314 W314
ANDW(034) A353 #FF00 W310
/U(432) W310 &256 W310
BIN(023) W310 W310
+(400) W310 &2000 W310
ANDW(034) A353 #FF W311
BIN(023) W311 W311

